FUNCTION "HF3_CP340_FC4301" : VOID	// FC 4301
TITLE = 配置本端所有CP340模块
//1：硬件配置 设置协议、波特率、奇偶校验位、起始地址
//2：需授权
//3：注意起始地址、DB块号（暂未填写）
VERSION : 0.1
BEGIN
NETWORK
TITLE = BA-21 电梯 H420/01(N) 672 2001~2005
      A     "Always0";
      =     L 0.0;
      BLD   103;
      A     "Always1";
      =     L 0.1;
      BLD   103;
      BLD   3;
      =     L 5.0;
      CDB;
      OPN   DI 1071;
      TAR2  LD 1;
      L     672;
      T     DIW 0;
      A     L 0.0;
      =     DIX 4.0;
      L     B#16#4A;
      T     DIB 5;
      L     31001;
      T     DIW 6;
      L     5;
      T     DIW 8;
      L     L#500;
      T     DID 10;
      A     L 0.1;
      =     DIX 14.0;
      L     2001;
      T     DIW 16;
      BLD   11;
      L     W#16#1002;
      T     LW 8;
      L     10;
      T     LW 10;
      L     30;
      T     LW 12;
      L     P#DBX 0.0;
      T     LD 14;
      L     W#16#1002;
      T     LW 18;
      L     10;
      T     LW 20;
      L     1071;
      T     LW 22;
      L     P#DBX 18.0;
      T     LD 24;
      UC    "BLKMOV";
      {     P#L 8.0, P#L 6.0, P#L 18.0 };
      BLD   11;
      L     W#16#1002;
      T     LW 8;
      L     10;
      T     LW 10;
      L     30;
      T     LW 12;
      L     P#DBX 10.0;
      T     LD 14;
      L     W#16#1002;
      T     LW 18;
      L     10;
      T     LW 20;
      L     1071;
      T     LW 22;
      L     P#DBX 28.0;
      T     LD 24;
      UC    "BLKMOV";
      {     P#L 8.0, P#L 6.0, P#L 18.0 };
      LAR2  P#DBX 0.0;
      UC    "MODMAS_STEP7_CP340_L";
      LAR2  LD 1;
      A     DIX 38.0;
      =     M 10.0;
      L     DIW 40;
      T     MW 12;
      L     DIW 42;
      T     MW 14;
      CDB;
      BLD   4;
      NOP   0;
NETWORK
TITLE = BA-21 局部排水泵 AP-PSB-B 688  2011~2015
      A     "Always0";
      =     L 0.0;
      BLD   103;
      A     "Always1";
      =     L 0.1;
      BLD   103;
      BLD   3;
      =     L 5.0;
      CDB;
      OPN   DI 1072;
      TAR2  LD 1;
      L     688;
      T     DIW 0;
      A     L 0.0;
      =     DIX 4.0;
      L     B#16#4A;
      T     DIB 5;
      L     31001;
      T     DIW 6;
      L     5;
      T     DIW 8;
      L     L#500;
      T     DID 10;
      A     L 0.1;
      =     DIX 14.0;
      L     2011;
      T     DIW 16;
      BLD   11;
      L     W#16#1002;
      T     LW 8;
      L     10;
      T     LW 10;
      L     30;
      T     LW 12;
      L     P#DBX 0.0;
      T     LD 14;
      L     W#16#1002;
      T     LW 18;
      L     10;
      T     LW 20;
      L     1072;
      T     LW 22;
      L     P#DBX 18.0;
      T     LD 24;
      UC    "BLKMOV";
      {     P#L 8.0, P#L 6.0, P#L 18.0 };
      BLD   11;
      L     W#16#1002;
      T     LW 8;
      L     10;
      T     LW 10;
      L     30;
      T     LW 12;
      L     P#DBX 10.0;
      T     LD 14;
      L     W#16#1002;
      T     LW 18;
      L     10;
      T     LW 20;
      L     1072;
      T     LW 22;
      L     P#DBX 28.0;
      T     LD 24;
      UC    "BLKMOV";
      {     P#L 8.0, P#L 6.0, P#L 18.0 };
      LAR2  P#DBX 0.0;
      UC    "MODMAS_STEP7_CP340_L";
      LAR2  LD 1;
      A     DIX 38.0;
      =     M 10.0;
      L     DIW 40;
      T     MW 12;
      L     DIW 42;
      T     MW 14;
      CDB;
      BLD   4;
      NOP   0;
NETWORK
TITLE = BA-21 自动扶梯 E420/05(K2)，E420/06(K2) 704 2021~2025
      A     "Always0";
      =     L 0.0;
      BLD   103;
      A     "Always1";
      =     L 0.1;
      BLD   103;
      BLD   3;
      =     L 5.0;
      CDB;
      OPN   DI 1073;
      TAR2  LD 1;
      L     704;
      T     DIW 0;
      A     L 0.0;
      =     DIX 4.0;
      L     B#16#4A;
      T     DIB 5;
      L     31001;
      T     DIW 6;
      L     5;
      T     DIW 8;
      L     L#500;
      T     DID 10;
      A     L 0.1;
      =     DIX 14.0;
      L     2021;
      T     DIW 16;
      BLD   11;
      L     W#16#1002;
      T     LW 8;
      L     10;
      T     LW 10;
      L     30;
      T     LW 12;
      L     P#DBX 0.0;
      T     LD 14;
      L     W#16#1002;
      T     LW 18;
      L     10;
      T     LW 20;
      L     1073;
      T     LW 22;
      L     P#DBX 18.0;
      T     LD 24;
      UC    "BLKMOV";
      {     P#L 8.0, P#L 6.0, P#L 18.0 };
      BLD   11;
      L     W#16#1002;
      T     LW 8;
      L     10;
      T     LW 10;
      L     30;
      T     LW 12;
      L     P#DBX 10.0;
      T     LD 14;
      L     W#16#1002;
      T     LW 18;
      L     10;
      T     LW 20;
      L     1073;
      T     LW 22;
      L     P#DBX 28.0;
      T     LD 24;
      UC    "BLKMOV";
      {     P#L 8.0, P#L 6.0, P#L 18.0 };
      LAR2  P#DBX 0.0;
      UC    "MODMAS_STEP7_CP340_L";
      LAR2  LD 1;
      A     DIX 38.0;
      =     M 10.0;
      L     DIW 40;
      T     MW 12;
      L     DIW 42;
      T     MW 14;
      CDB;
      BLD   4;
      NOP   0;
NETWORK
TITLE = BA-21 不间断电源 UPS-1 720 2031~2035
      A     "Always0";
      =     L 0.0;
      BLD   103;
      A     "Always1";
      =     L 0.1;
      BLD   103;
      BLD   3;
      =     L 5.0;
      CDB;
      OPN   DI 1074;
      TAR2  LD 1;
      L     720;
      T     DIW 0;
      A     L 0.0;
      =     DIX 4.0;
      L     B#16#4A;
      T     DIB 5;
      L     31001;
      T     DIW 6;
      L     5;
      T     DIW 8;
      L     L#500;
      T     DID 10;
      A     L 0.1;
      =     DIX 14.0;
      L     2031;
      T     DIW 16;
      BLD   11;
      L     W#16#1002;
      T     LW 8;
      L     10;
      T     LW 10;
      L     30;
      T     LW 12;
      L     P#DBX 0.0;
      T     LD 14;
      L     W#16#1002;
      T     LW 18;
      L     10;
      T     LW 20;
      L     1074;
      T     LW 22;
      L     P#DBX 18.0;
      T     LD 24;
      UC    "BLKMOV";
      {     P#L 8.0, P#L 6.0, P#L 18.0 };
      BLD   11;
      L     W#16#1002;
      T     LW 8;
      L     10;
      T     LW 10;
      L     30;
      T     LW 12;
      L     P#DBX 10.0;
      T     LD 14;
      L     W#16#1002;
      T     LW 18;
      L     10;
      T     LW 20;
      L     1074;
      T     LW 22;
      L     P#DBX 28.0;
      T     LD 24;
      UC    "BLKMOV";
      {     P#L 8.0, P#L 6.0, P#L 18.0 };
      LAR2  P#DBX 0.0;
      UC    "MODMAS_STEP7_CP340_L";
      LAR2  LD 1;
      A     DIX 38.0;
      =     M 10.0;
      L     DIW 40;
      T     MW 12;
      L     DIW 42;
      T     MW 14;
      CDB;
      BLD   4;
      NOP   0;
NETWORK
TITLE = BA-22 应急照明 EPS21 736 2041~2045
      A     "Always0";
      =     L 0.0;
      BLD   103;
      A     "Always1";
      =     L 0.1;
      BLD   103;
      BLD   3;
      =     L 5.0;
      CDB;
      OPN   DI 1075;
      TAR2  LD 1;
      L     736;
      T     DIW 0;
      A     L 0.0;
      =     DIX 4.0;
      L     B#16#4A;
      T     DIB 5;
      L     31001;
      T     DIW 6;
      L     5;
      T     DIW 8;
      L     L#500;
      T     DID 10;
      A     L 0.1;
      =     DIX 14.0;
      L     2041;
      T     DIW 16;
      BLD   11;
      L     W#16#1002;
      T     LW 8;
      L     10;
      T     LW 10;
      L     30;
      T     LW 12;
      L     P#DBX 0.0;
      T     LD 14;
      L     W#16#1002;
      T     LW 18;
      L     10;
      T     LW 20;
      L     1075;
      T     LW 22;
      L     P#DBX 18.0;
      T     LD 24;
      UC    "BLKMOV";
      {     P#L 8.0, P#L 6.0, P#L 18.0 };
      BLD   11;
      L     W#16#1002;
      T     LW 8;
      L     10;
      T     LW 10;
      L     30;
      T     LW 12;
      L     P#DBX 10.0;
      T     LD 14;
      L     W#16#1002;
      T     LW 18;
      L     10;
      T     LW 20;
      L     1075;
      T     LW 22;
      L     P#DBX 28.0;
      T     LD 24;
      UC    "BLKMOV";
      {     P#L 8.0, P#L 6.0, P#L 18.0 };
      LAR2  P#DBX 0.0;
      UC    "MODMAS_STEP7_CP340_L";
      LAR2  LD 1;
      A     DIX 38.0;
      =     M 10.0;
      L     DIW 40;
      T     MW 12;
      L     DIW 42;
      T     MW 14;
      CDB;
      BLD   4;
      NOP   0;
NETWORK
TITLE = BA-22 雨水泵 AT-AYSB1，AT-AYSB2 752 2051~2055
      A     "Always0";
      =     L 0.0;
      BLD   103;
      A     "Always1";
      =     L 0.1;
      BLD   103;
      BLD   3;
      =     L 5.0;
      CDB;
      OPN   DI 1076;
      TAR2  LD 1;
      L     752;
      T     DIW 0;
      A     L 0.0;
      =     DIX 4.0;
      L     B#16#4A;
      T     DIB 5;
      L     31001;
      T     DIW 6;
      L     5;
      T     DIW 8;
      L     L#500;
      T     DID 10;
      A     L 0.1;
      =     DIX 14.0;
      L     2051;
      T     DIW 16;
      BLD   11;
      L     W#16#1002;
      T     LW 8;
      L     10;
      T     LW 10;
      L     30;
      T     LW 12;
      L     P#DBX 0.0;
      T     LD 14;
      L     W#16#1002;
      T     LW 18;
      L     10;
      T     LW 20;
      L     1076;
      T     LW 22;
      L     P#DBX 18.0;
      T     LD 24;
      UC    "BLKMOV";
      {     P#L 8.0, P#L 6.0, P#L 18.0 };
      BLD   11;
      L     W#16#1002;
      T     LW 8;
      L     10;
      T     LW 10;
      L     30;
      T     LW 12;
      L     P#DBX 10.0;
      T     LD 14;
      L     W#16#1002;
      T     LW 18;
      L     10;
      T     LW 20;
      L     1076;
      T     LW 22;
      L     P#DBX 28.0;
      T     LD 24;
      UC    "BLKMOV";
      {     P#L 8.0, P#L 6.0, P#L 18.0 };
      LAR2  P#DBX 0.0;
      UC    "MODMAS_STEP7_CP340_L";
      LAR2  LD 1;
      A     DIX 38.0;
      =     M 10.0;
      L     DIW 40;
      T     MW 12;
      L     DIW 42;
      T     MW 14;
      CDB;
      BLD   4;
      NOP   0;
NETWORK
TITLE = BA-22 雨水泵 AT-AYSB3，AT-AYSB4，AP-FSB2 768  2061~2065
      A     "Always0";
      =     L 0.0;
      BLD   103;
      A     "Always1";
      =     L 0.1;
      BLD   103;
      BLD   3;
      =     L 5.0;
      CDB;
      OPN   DI 1077;
      TAR2  LD 1;
      L     768;
      T     DIW 0;
      A     L 0.0;
      =     DIX 4.0;
      L     B#16#4A;
      T     DIB 5;
      L     31001;
      T     DIW 6;
      L     5;
      T     DIW 8;
      L     L#500;
      T     DID 10;
      A     L 0.1;
      =     DIX 14.0;
      L     2061;
      T     DIW 16;
      BLD   11;
      L     W#16#1002;
      T     LW 8;
      L     10;
      T     LW 10;
      L     30;
      T     LW 12;
      L     P#DBX 0.0;
      T     LD 14;
      L     W#16#1002;
      T     LW 18;
      L     10;
      T     LW 20;
      L     1077;
      T     LW 22;
      L     P#DBX 18.0;
      T     LD 24;
      UC    "BLKMOV";
      {     P#L 8.0, P#L 6.0, P#L 18.0 };
      BLD   11;
      L     W#16#1002;
      T     LW 8;
      L     10;
      T     LW 10;
      L     30;
      T     LW 12;
      L     P#DBX 10.0;
      T     LD 14;
      L     W#16#1002;
      T     LW 18;
      L     10;
      T     LW 20;
      L     1077;
      T     LW 22;
      L     P#DBX 28.0;
      T     LD 24;
      UC    "BLKMOV";
      {     P#L 8.0, P#L 6.0, P#L 18.0 };
      LAR2  P#DBX 0.0;
      UC    "MODMAS_STEP7_CP340_L";
      LAR2  LD 1;
      A     DIX 38.0;
      =     M 10.0;
      L     DIW 40;
      T     MW 12;
      L     DIW 42;
      T     MW 14;
      CDB;
      BLD   4;
      NOP   0;
NETWORK
TITLE = BA-22 局排废水泵 AP-PSB-C 784 2071~2075
      A     "Always0";
      =     L 0.0;
      BLD   103;
      A     "Always1";
      =     L 0.1;
      BLD   103;
      BLD   3;
      =     L 5.0;
      CDB;
      OPN   DI 1078;
      TAR2  LD 1;
      L     784;
      T     DIW 0;
      A     L 0.0;
      =     DIX 4.0;
      L     B#16#4A;
      T     DIB 5;
      L     31001;
      T     DIW 6;
      L     5;
      T     DIW 8;
      L     L#500;
      T     DID 10;
      A     L 0.1;
      =     DIX 14.0;
      L     2071;
      T     DIW 16;
      BLD   11;
      L     W#16#1002;
      T     LW 8;
      L     10;
      T     LW 10;
      L     30;
      T     LW 12;
      L     P#DBX 0.0;
      T     LD 14;
      L     W#16#1002;
      T     LW 18;
      L     10;
      T     LW 20;
      L     1078;
      T     LW 22;
      L     P#DBX 18.0;
      T     LD 24;
      UC    "BLKMOV";
      {     P#L 8.0, P#L 6.0, P#L 18.0 };
      BLD   11;
      L     W#16#1002;
      T     LW 8;
      L     10;
      T     LW 10;
      L     30;
      T     LW 12;
      L     P#DBX 10.0;
      T     LD 14;
      L     W#16#1002;
      T     LW 18;
      L     10;
      T     LW 20;
      L     1078;
      T     LW 22;
      L     P#DBX 28.0;
      T     LD 24;
      UC    "BLKMOV";
      {     P#L 8.0, P#L 6.0, P#L 18.0 };
      LAR2  P#DBX 0.0;
      UC    "MODMAS_STEP7_CP340_L";
      LAR2  LD 1;
      A     DIX 38.0;
      =     M 10.0;
      L     DIW 40;
      T     MW 12;
      L     DIW 42;
      T     MW 14;
      CDB;
      BLD   4;
      NOP   0;
NETWORK
TITLE = BA-22 自动扶梯 E420/07(K3) 800 2081~2085
      A     "Always0";
      =     L 0.0;
      BLD   103;
      A     "Always1";
      =     L 0.1;
      BLD   103;
      BLD   3;
      =     L 5.0;
      CDB;
      OPN   DI 1079;
      TAR2  LD 1;
      L     800;
      T     DIW 0;
      A     L 0.0;
      =     DIX 4.0;
      L     B#16#4A;
      T     DIB 5;
      L     31001;
      T     DIW 6;
      L     5;
      T     DIW 8;
      L     L#500;
      T     DID 10;
      A     L 0.1;
      =     DIX 14.0;
      L     2081;
      T     DIW 16;
      BLD   11;
      L     W#16#1002;
      T     LW 8;
      L     10;
      T     LW 10;
      L     30;
      T     LW 12;
      L     P#DBX 0.0;
      T     LD 14;
      L     W#16#1002;
      T     LW 18;
      L     10;
      T     LW 20;
      L     1079;
      T     LW 22;
      L     P#DBX 18.0;
      T     LD 24;
      UC    "BLKMOV";
      {     P#L 8.0, P#L 6.0, P#L 18.0 };
      BLD   11;
      L     W#16#1002;
      T     LW 8;
      L     10;
      T     LW 10;
      L     30;
      T     LW 12;
      L     P#DBX 10.0;
      T     LD 14;
      L     W#16#1002;
      T     LW 18;
      L     10;
      T     LW 20;
      L     1079;
      T     LW 22;
      L     P#DBX 28.0;
      T     LD 24;
      UC    "BLKMOV";
      {     P#L 8.0, P#L 6.0, P#L 18.0 };
      LAR2  P#DBX 0.0;
      UC    "MODMAS_STEP7_CP340_L";
      LAR2  LD 1;
      A     DIX 38.0;
      =     M 10.0;
      L     DIW 40;
      T     MW 12;
      L     DIW 42;
      T     MW 14;
      CDB;
      BLD   4;
      NOP   0;
NETWORK
TITLE = BA-11 应急照明 EPS11 816 2091~2095
      A     "Always0";
      =     L 0.0;
      BLD   103;
      A     "Always1";
      =     L 0.1;
      BLD   103;
      BLD   3;
      =     L 5.0;
      CDB;
      OPN   DI 1080;
      TAR2  LD 1;
      L     816;
      T     DIW 0;
      A     L 0.0;
      =     DIX 4.0;
      L     B#16#4A;
      T     DIB 5;
      L     31001;
      T     DIW 6;
      L     5;
      T     DIW 8;
      L     L#500;
      T     DID 10;
      A     L 0.1;
      =     DIX 14.0;
      L     2091;
      T     DIW 16;
      BLD   11;
      L     W#16#1002;
      T     LW 8;
      L     10;
      T     LW 10;
      L     30;
      T     LW 12;
      L     P#DBX 0.0;
      T     LD 14;
      L     W#16#1002;
      T     LW 18;
      L     10;
      T     LW 20;
      L     1080;
      T     LW 22;
      L     P#DBX 18.0;
      T     LD 24;
      UC    "BLKMOV";
      {     P#L 8.0, P#L 6.0, P#L 18.0 };
      BLD   11;
      L     W#16#1002;
      T     LW 8;
      L     10;
      T     LW 10;
      L     30;
      T     LW 12;
      L     P#DBX 10.0;
      T     LD 14;
      L     W#16#1002;
      T     LW 18;
      L     10;
      T     LW 20;
      L     1080;
      T     LW 22;
      L     P#DBX 28.0;
      T     LD 24;
      UC    "BLKMOV";
      {     P#L 8.0, P#L 6.0, P#L 18.0 };
      LAR2  P#DBX 0.0;
      UC    "MODMAS_STEP7_CP340_L";
      LAR2  LD 1;
      A     DIX 38.0;
      =     M 10.0;
      L     DIW 40;
      T     MW 12;
      L     DIW 42;
      T     MW 14;
      CDB;
      BLD   4;
      NOP   0;
NETWORK
TITLE = BA-11 自动扶梯 E420/01(N) 832 2101~2105
      A     "Always0";
      =     L 0.0;
      BLD   103;
      A     "Always1";
      =     L 0.1;
      BLD   103;
      BLD   3;
      =     L 5.0;
      CDB;
      OPN   DI 1081;
      TAR2  LD 1;
      L     832;
      T     DIW 0;
      A     L 0.0;
      =     DIX 4.0;
      L     B#16#4A;
      T     DIB 5;
      L     31001;
      T     DIW 6;
      L     5;
      T     DIW 8;
      L     L#500;
      T     DID 10;
      A     L 0.1;
      =     DIX 14.0;
      L     2101;
      T     DIW 16;
      BLD   11;
      L     W#16#1002;
      T     LW 8;
      L     10;
      T     LW 10;
      L     30;
      T     LW 12;
      L     P#DBX 0.0;
      T     LD 14;
      L     W#16#1002;
      T     LW 18;
      L     10;
      T     LW 20;
      L     1081;
      T     LW 22;
      L     P#DBX 18.0;
      T     LD 24;
      UC    "BLKMOV";
      {     P#L 8.0, P#L 6.0, P#L 18.0 };
      BLD   11;
      L     W#16#1002;
      T     LW 8;
      L     10;
      T     LW 10;
      L     30;
      T     LW 12;
      L     P#DBX 10.0;
      T     LD 14;
      L     W#16#1002;
      T     LW 18;
      L     10;
      T     LW 20;
      L     1081;
      T     LW 22;
      L     P#DBX 28.0;
      T     LD 24;
      UC    "BLKMOV";
      {     P#L 8.0, P#L 6.0, P#L 18.0 };
      LAR2  P#DBX 0.0;
      UC    "MODMAS_STEP7_CP340_L";
      LAR2  LD 1;
      A     DIX 38.0;
      =     M 10.0;
      L     DIW 40;
      T     MW 12;
      L     DIW 42;
      T     MW 14;
      CDB;
      BLD   4;
      NOP   0;
NETWORK
TITLE = BQ11 区间水泵 ATD-HSB 944 2181~2185
      A     "Always0";
      =     L 0.0;
      BLD   103;
      A     "Always1";
      =     L 0.1;
      BLD   103;
      BLD   3;
      =     L 5.0;
      CDB;
      OPN   DI 1082;
      TAR2  LD 1;
      L     944;
      T     DIW 0;
      A     L 0.0;
      =     DIX 4.0;
      L     B#16#4A;
      T     DIB 5;
      L     31001;
      T     DIW 6;
      L     5;
      T     DIW 8;
      L     L#500;
      T     DID 10;
      A     L 0.1;
      =     DIX 14.0;
      L     2181;
      T     DIW 16;
      BLD   11;
      L     W#16#1002;
      T     LW 8;
      L     10;
      T     LW 10;
      L     30;
      T     LW 12;
      L     P#DBX 0.0;
      T     LD 14;
      L     W#16#1002;
      T     LW 18;
      L     10;
      T     LW 20;
      L     1082;
      T     LW 22;
      L     P#DBX 18.0;
      T     LD 24;
      UC    "BLKMOV";
      {     P#L 8.0, P#L 6.0, P#L 18.0 };
      BLD   11;
      L     W#16#1002;
      T     LW 8;
      L     10;
      T     LW 10;
      L     30;
      T     LW 12;
      L     P#DBX 10.0;
      T     LD 14;
      L     W#16#1002;
      T     LW 18;
      L     10;
      T     LW 20;
      L     1082;
      T     LW 22;
      L     P#DBX 28.0;
      T     LD 24;
      UC    "BLKMOV";
      {     P#L 8.0, P#L 6.0, P#L 18.0 };
      LAR2  P#DBX 0.0;
      UC    "MODMAS_STEP7_CP340_L";
      LAR2  LD 1;
      A     DIX 38.0;
      =     M 10.0;
      L     DIW 40;
      T     MW 12;
      L     DIW 42;
      T     MW 14;
      CDB;
      BLD   4;
      NOP   0;
END_FUNCTION

DATA_BLOCK "CONTROL_DAT"	// DB 1
VERSION : 0.1
  STRUCT
   id_0_a : WORD ;
   id_1_a : WORD ;
   reuse_conn_time : TIME ;
   use_all_conn : BOOL ;
   RECV_TIMEOUT : TIME ;
   CONN_TIMEOUT : TIME ;
   DISCONNECT : BOOL ;
   Init : BOOL ;
   ENQ : BOOL ;
   DATA_TYPE : BYTE ;
   START_ADDRESS : WORD ;
   LENGTH : WORD ;
   WRITE_READ : BOOL ;
   UNIT : BYTE  := B#16#1;
   LICENSED : BOOL ;
   BUSY : BOOL ;
   DONE : BOOL ;
   ERROR : BOOL ;
   ESTAB_0A : BOOL ;
   STATUS_0A : WORD ;
   ESTAB_1A : BOOL ;
   STATUS_1A : WORD ;
   RedErrS7 : BOOL ;
   RedErrDev : BOOL ;
   TotComErr : BOOL ;
   Init_Error : BOOL ;
   Init_Status : WORD ;
   Save_STATUS_0A : WORD ;
   Save_STATUS_1A : WORD ;
   Count_Done : DINT ;
   Count_Error : DINT ;
  END_STRUCT ;	
BEGIN
   UNIT := B#16#1;
END_DATA_BLOCK

DATA_BLOCK "MODBUS_HPARAM_PN_2"	// DB 2
TITLE = Parameters for Modbus TCP
AUTHOR : SIEMENS
FAMILY : COMM
NAME : MBHPARAM
VERSION : 0.1
  STRUCT
   double_sided_red : BOOL ;
   connection_0A : STRUCT
    block_length : WORD  := W#16#40;	//#!Verbindung_0001!#
    id : WORD  := W#16#1;
    connection_type : BYTE  := B#16#11;
    active_est : BOOL  := TRUE;
    local_device_id : BYTE  := B#16#5;
    local_tsap_id_len : BYTE ;
    rem_subnet_id_len : BYTE ;
    rem_staddr_len : BYTE  := B#16#4;
    rem_tsap_id_len : BYTE  := B#16#2;
    next_staddr_len : BYTE ;
    local_tsap_id : ARRAY  [1 .. 16 ] OF BYTE  := 16 (B#16#0) ;
    rem_subnet_id : ARRAY  [1 .. 6 ] OF BYTE  := B#16#0, B#16#0, B#16#0, B#16#0, B#16#0, B#16#0;
    rem_staddr : ARRAY  [1 .. 6 ] OF BYTE  := B#16#A, B#16#2E, B#16#1E, B#16#97;
    rem_tsap_id : ARRAY  [1 .. 16 ] OF BYTE  := B#16#1, B#16#F6;
    next_staddr : ARRAY  [1 .. 6 ] OF BYTE  := B#16#0, B#16#0, B#16#0, B#16#0, B#16#0, B#16#0;
    spare : WORD ;	//#!Verbindung_0001!#
   END_STRUCT ;
   connection_1A : STRUCT
    block_length : WORD  := W#16#40;	//#!Verbindung_0002!#
    id : WORD  := W#16#2;
    connection_type : BYTE  := B#16#11;
    active_est : BOOL  := TRUE;
    local_device_id : BYTE  := B#16#15;
    local_tsap_id_len : BYTE ;
    rem_subnet_id_len : BYTE ;
    rem_staddr_len : BYTE  := B#16#4;
    rem_tsap_id_len : BYTE  := B#16#2;
    next_staddr_len : BYTE ;
    local_tsap_id : ARRAY  [1 .. 16 ] OF BYTE  := 16 (B#16#0) ;
    rem_subnet_id : ARRAY  [1 .. 6 ] OF BYTE  := B#16#0, B#16#0, B#16#0, B#16#0, B#16#0, B#16#0;
    rem_staddr : ARRAY  [1 .. 6 ] OF BYTE  := B#16#A, B#16#2E, B#16#82, B#16#97;
    rem_tsap_id : ARRAY  [1 .. 16 ] OF BYTE  := B#16#1, B#16#F6;
    next_staddr : ARRAY  [1 .. 6 ] OF BYTE  := B#16#0, B#16#0, B#16#0, B#16#0, B#16#0, B#16#0;
    spare : WORD ;	//#!Verbindung_0002!#
   END_STRUCT ;
   server_client : BOOL ;
   single_write : BOOL ;
   connect_at_startup : BOOL  := TRUE;
   reserved : BYTE ;
   data_type_1 : BYTE  := B#16#3;
   db_1 : WORD  := W#16#8F3;
   start_1 : WORD ;
   end_1 : WORD  := W#16#18F;
   data_type_2 : BYTE  := B#16#3;
   db_2 : WORD  := W#16#8F4;
   start_2 : WORD  := W#16#190;
   end_2 : WORD  := W#16#22F;
   data_type_3 : BYTE ;
   db_3 : WORD  := W#16#D;
   start_3 : WORD  := W#16#2D0;
   end_3 : WORD  := W#16#3E8;
   data_type_4 : BYTE ;
   db_4 : WORD ;
   start_4 : WORD ;
   end_4 : WORD ;
   data_type_5 : BYTE ;
   db_5 : WORD  := W#16#E;
   start_5 : WORD  := W#16#280;
   end_5 : WORD  := W#16#4E2;
   data_type_6 : BYTE ;
   db_6 : WORD  := W#16#F;
   start_6 : WORD  := W#16#6A4;
   end_6 : WORD  := W#16#8FC;
   data_type_7 : BYTE ;
   db_7 : WORD  := W#16#10;
   start_7 : WORD  := W#16#6A4;
   end_7 : WORD  := W#16#8FC;
   data_type_8 : BYTE ;
   db_8 : WORD ;
   start_8 : WORD ;
   end_8 : WORD ;
   conn_0A_send_buffer : ARRAY  [1 .. 260 ] OF BYTE  := 260 (B#16#0) ;
   conn_0A_recv_buffer : ARRAY  [1 .. 260 ] OF BYTE  := 260 (B#16#0) ;
   conn_1A_send_buffer : ARRAY  [1 .. 260 ] OF BYTE  := 260 (B#16#0) ;
   conn_1A_recv_buffer : ARRAY  [1 .. 260 ] OF BYTE  := 260 (B#16#0) ;
  END_STRUCT ;	
BEGIN
   connection_0A.block_length := W#16#40;
   connection_0A.id := W#16#1;
   connection_0A.connection_type := B#16#11;
   connection_0A.active_est := TRUE;
   connection_0A.local_device_id := B#16#5;
   connection_0A.rem_staddr_len := B#16#4;
   connection_0A.rem_tsap_id_len := B#16#2;
   connection_0A.rem_staddr[1] := B#16#A;
   connection_0A.rem_staddr[2] := B#16#2E;
   connection_0A.rem_staddr[3] := B#16#1E;
   connection_0A.rem_staddr[4] := B#16#97;
   connection_0A.rem_tsap_id[1] := B#16#1;
   connection_0A.rem_tsap_id[2] := B#16#F6;
   connection_1A.block_length := W#16#40;
   connection_1A.id := W#16#2;
   connection_1A.connection_type := B#16#11;
   connection_1A.active_est := TRUE;
   connection_1A.local_device_id := B#16#15;
   connection_1A.rem_staddr_len := B#16#4;
   connection_1A.rem_tsap_id_len := B#16#2;
   connection_1A.rem_staddr[1] := B#16#A;
   connection_1A.rem_staddr[2] := B#16#2E;
   connection_1A.rem_staddr[3] := B#16#82;
   connection_1A.rem_staddr[4] := B#16#97;
   connection_1A.rem_tsap_id[1] := B#16#1;
   connection_1A.rem_tsap_id[2] := B#16#F6;
   connect_at_startup := TRUE;
   data_type_1 := B#16#3;
   db_1 := W#16#8F3;
   end_1 := W#16#18F;
   data_type_2 := B#16#3;
   db_2 := W#16#8F4;
   start_2 := W#16#190;
   end_2 := W#16#22F;
   db_3 := W#16#D;
   start_3 := W#16#2D0;
   end_3 := W#16#3E8;
   db_5 := W#16#E;
   start_5 := W#16#280;
   end_5 := W#16#4E2;
   db_6 := W#16#F;
   start_6 := W#16#6A4;
   end_6 := W#16#8FC;
   db_7 := W#16#10;
   start_7 := W#16#6A4;
   end_7 := W#16#8FC;
END_DATA_BLOCK

DATA_BLOCK "License DB"	// DB 3
VERSION : 0.1
  STRUCT
   REG_KEY : STRING  [17 ] := 'insert REG_KEY';	//Registration Key
  END_STRUCT ;	
BEGIN
   REG_KEY := 'insert REG_KEY';
END_DATA_BLOCK

DATA_BLOCK DB 10
VERSION : 0.1
  STRUCT
   DB_VAR1 : REAL  := 6.700000e+000;	//Temporary placeholder variable
   DB_VAR2 : REAL ;
  END_STRUCT ;	
BEGIN
END_DATA_BLOCK

DATA_BLOCK DB 12
VERSION : 0.1
  STRUCT
   DB_VAR : ARRAY  [0 .. 76 ] OF //Holding Register 3001-3077
   WORD  := 77 (W#16#0) ;
   reserved : WORD ;
  END_STRUCT ;	
BEGIN
END_DATA_BLOCK

DATA_BLOCK "CPULINDB"	// DB 30
VERSION : 0.1
  STRUCT
   YOULIN1 : STRING  [8 ] := 'R1R3H5Y4';	//Temporary placeholder variable
   YOULIN2 : STRING  [8 ] := '3N5L1J32';
  END_STRUCT ;	
BEGIN
   YOULIN1 := 'R1R3H5Y4';
   YOULIN2 := '3N5L1J32';
END_DATA_BLOCK

DATA_BLOCK "SYS_Date_Time_D"	// DB 34
VERSION : 0.1
  STRUCT
   SET_DATE_TIME : ARRAY  [1 .. 8 ] OF //年月日时分秒
   BYTE ;
   READ_DATE_TIME : ARRAY  [1 .. 8 ] OF BYTE ;
   SET : DATE_AND_TIME ;
   READ : DATE_AND_TIME ;
   TIME_HM : INT ;	//时分(2359表示23点59分)
  END_STRUCT ;	
BEGIN
END_DATA_BLOCK

DATA_BLOCK "FB200_DB"	// DB 200
VERSION : 0.0
"S7400H-COM-MAIN-SLAVE"
BEGIN
END_DATA_BLOCK

DATA_BLOCK "FB201_DB"	// DB 201
VERSION : 0.0
"S7400H-COM-MAIN-IBP"
BEGIN
END_DATA_BLOCK

DATA_BLOCK "MAIN-READ-SLAVE"	// DB 202
VERSION : 0.1
  STRUCT
   MAIN_R_SLAVE : ARRAY  [0 .. 4000 ] OF //Temporary placeholder variable
   INT  := 0;
  END_STRUCT ;	
BEGIN
END_DATA_BLOCK

DATA_BLOCK "MAIN-WRITE-SLAVE"	// DB 203
VERSION : 0.1
  STRUCT
   MAIN_W_SLAVE : ARRAY  [0 .. 4000 ] OF //Temporary placeholder variable
   INT  := 0;
  END_STRUCT ;	
BEGIN
END_DATA_BLOCK

DATA_BLOCK "MAIN-READ-IBP"	// DB 204
VERSION : 0.1
  STRUCT
   MAIN_R_IBP : ARRAY  [0 .. 4000 ] OF //Temporary placeholder variable
   INT  := 0;
  END_STRUCT ;	
BEGIN
END_DATA_BLOCK

DATA_BLOCK "MAIN-WRITE-IBP"	// DB 205
VERSION : 0.1
  STRUCT
   MAIN_W_IBP : ARRAY  [0 .. 4000 ] OF //Temporary placeholder variable
   INT  := 0;
  END_STRUCT ;	
BEGIN
END_DATA_BLOCK

DATA_BLOCK "DETAIL_DIAG_DB_RACK0"	// DB 458
AUTHOR : SIEMENS
FAMILY : DP
VERSION : 0.1
"DETAIL_DP_DIAG"
BEGIN
END_DATA_BLOCK

DATA_BLOCK "DETAIL_DIAG_DB_RACK1"	// DB 459
AUTHOR : SIEMENS
FAMILY : DP
VERSION : 0.1
"DETAIL_DP_DIAG"
BEGIN
END_DATA_BLOCK

DATA_BLOCK "DP_ERROR_RACK0"	// DB 460
VERSION : 0.1
  STRUCT
   STATE : ARRAY  [0 .. 500 ] OF //Temporary placeholder variable
   INT ;
   STATE_NONE : ARRAY  [0 .. 50 ] OF INT ;
   ALL_OK : BOOL ;
   TIME_RESET : BOOL ;
   NOTUSED : ARRAY  [0 .. 250 ] OF INT ;
  END_STRUCT ;	
BEGIN
END_DATA_BLOCK

DATA_BLOCK "DP_ERROR_RESET_DB"	// DB 461
VERSION : 0.1
  STRUCT
   STATE : ARRAY  [0 .. 500 ] OF //Temporary placeholder variable
   INT ;
   STATE_NONE : ARRAY  [0 .. 50 ] OF INT ;
   ALL_OK : BOOL ;
   TIME_RESET : BOOL ;
   NOTUSED : ARRAY  [0 .. 250 ] OF INT ;
  END_STRUCT ;	
BEGIN
END_DATA_BLOCK

DATA_BLOCK "DP_ERROR_FB1501"	// DB 462
VERSION : 0.0
"com_check"
BEGIN
END_DATA_BLOCK

DATA_BLOCK "DB_FOR_FB300"	// DB 463
VERSION : 0.1
"READ_ERROR"
BEGIN
END_DATA_BLOCK

DATA_BLOCK "DP_VAT"	// DB 464
VERSION : 0.1
  STRUCT
   MANUAL_MODE : BOOL ;
   SINGLE_STEP_SLAVE : BOOL ;
   SINGLE_STEP_ERROR : BOOL ;
   RESET : BOOL ;
   SINGLE_SLAVE_DIAG : BOOL ;
   SINGLE_DIAG_ADR : BYTE ;
   ALL_SLAVES_OK : BOOL ;
   SUM_SLAVES_DIAG : BYTE ;
   SLAVE_ADR : BYTE ;
   SLAVE_STATE : BYTE ;
   SLAVE_IDENT_NO : WORD ;
   ERROR_NO : BYTE ;
   ERROR_TYPE : BYTE ;
   MODULE_NO : BYTE ;
   MODULE_STATE : BYTE ;
   CHANNEL_NO : BYTE ;
   CHANNEL_TYPE : BYTE ;
   CHANNEL_ERROR_CODE : INT ;
   CHANNEL_ERROR_INFO_1 : DWORD ;
   CHANNEL_ERROR_INFO_2 : DWORD ;
   DIAG_COUNTER : BYTE ;
   DIAG_OVERFLOW : BOOL ;
   BUSY : BOOL ;
   MANUAL_MODE1 : BOOL ;
   SINGLE_STEP_SLAVE1 : BOOL ;
   SINGLE_STEP_ERROR1 : BOOL ;
   RESET1 : BOOL ;
   SINGLE_SLAVE_DIAG1 : BOOL ;
   SINGLE_DIAG_ADR1 : BYTE ;
   ALL_SLAVES_OK1 : BOOL ;
   SUM_SLAVES_DIAG1 : BYTE ;
   SLAVE_ADR1 : BYTE ;
   SLAVE_STATE1 : BYTE ;
   SLAVE_IDENT_NO1 : WORD ;
   ERROR_NO1 : BYTE ;
   ERROR_TYPE1 : BYTE ;
   MODULE_NO1 : BYTE ;
   MODULE_STATE1 : BYTE ;
   CHANNEL_NO1 : BYTE ;
   CHANNEL_TYPE1 : BYTE ;
   CHANNEL_ERROR_CODE1 : INT ;
   CHANNEL_ERROR_INFO_11 : DWORD ;
   CHANNEL_ERROR_INFO_21 : DWORD ;
   DIAG_COUNTER1 : BYTE ;
   DIAG_OVERFLOW1 : BOOL ;
   BUSY1 : BOOL ;
   TIME_RESET : BOOL ;
  END_STRUCT ;	
BEGIN
END_DATA_BLOCK

DATA_BLOCK "DP_ERROR_RACK1"	// DB 465
VERSION : 0.1
  STRUCT
   STATE : ARRAY  [0 .. 500 ] OF //Temporary placeholder variable
   INT ;
   STATE_NONE : ARRAY  [0 .. 50 ] OF INT ;
   ALL_OK : BOOL ;
   TIME_RESET : BOOL ;
   NOTUSED : ARRAY  [0 .. 250 ] OF INT ;
  END_STRUCT ;	
BEGIN
END_DATA_BLOCK

DATA_BLOCK "DP_ERROR1_RESET"	// DB 466
VERSION : 0.1
  STRUCT
   STATE : ARRAY  [0 .. 500 ] OF //Temporary placeholder variable
   INT ;
   STATE_NONE : ARRAY  [0 .. 50 ] OF INT ;
   ALL_OK : BOOL ;
   TIME_RESET : BOOL ;
   NOTUSED : ARRAY  [0 .. 250 ] OF INT ;
  END_STRUCT ;	
BEGIN
END_DATA_BLOCK

DATA_BLOCK "DP_ERROR1_FB1501"	// DB 467
VERSION : 0.0
"com_check"
BEGIN
END_DATA_BLOCK

DATA_BLOCK "FB523_DB"	// DB 523
AUTHOR : KNAB
FAMILY : DIAGNOSE
VERSION : 0.0
"H_STATUS"
BEGIN
END_DATA_BLOCK

DATA_BLOCK "LED"	// DB 525
VERSION : 0.1
  STRUCT
   EXTF : ARRAY  [0 .. 8 ] OF BYTE ;
   REDF : ARRAY  [0 .. 8 ] OF BYTE ;
   EXTF_RET_VAL : INT ;
   REDF_RET_VAL : INT ;
   EXTF_BUSY : BOOL ;
   REDF_BUSY : BOOL ;
  END_STRUCT ;	
BEGIN
END_DATA_BLOCK

DATA_BLOCK DB 777
VERSION : 0.0
"HF4_IMCC_TVF_FB2652"
BEGIN
END_DATA_BLOCK

DATA_BLOCK "IDB_MODBUS"	// DB 915
AUTHOR : SIEMENS
FAMILY : COMM
VERSION : 0.0
"MB_PNHCL"
BEGIN
END_DATA_BLOCK

DATA_BLOCK "JOBLIST_DB"	// DB 919
AUTHOR : SIEMENS
FAMILY : COMM
VERSION : 0.0
"Job_List"
BEGIN
END_DATA_BLOCK

DATA_BLOCK "JOB_RESET_DB"	// DB 921
VERSION : 0.0
"JOB_RESET"
BEGIN
END_DATA_BLOCK

DATA_BLOCK DB 1072
AUTHOR : Dixinke
FAMILY : ASCMOD
VERSION : 0.0
"MODMAS_STEP7_CP340_L"
BEGIN
END_DATA_BLOCK

DATA_BLOCK DB 1073
AUTHOR : Dixinke
FAMILY : ASCMOD
VERSION : 0.0
"MODMAS_STEP7_CP340_L"
BEGIN
END_DATA_BLOCK

DATA_BLOCK DB 1074
AUTHOR : Dixinke
FAMILY : ASCMOD
VERSION : 0.0
"MODMAS_STEP7_CP340_L"
BEGIN
END_DATA_BLOCK

DATA_BLOCK DB 1075
AUTHOR : Dixinke
FAMILY : ASCMOD
VERSION : 0.0
"MODMAS_STEP7_CP340_L"
BEGIN
END_DATA_BLOCK

DATA_BLOCK DB 1076
AUTHOR : Dixinke
FAMILY : ASCMOD
VERSION : 0.0
"MODMAS_STEP7_CP340_L"
BEGIN
END_DATA_BLOCK

DATA_BLOCK DB 1077
AUTHOR : Dixinke
FAMILY : ASCMOD
VERSION : 0.0
"MODMAS_STEP7_CP340_L"
BEGIN
END_DATA_BLOCK

DATA_BLOCK DB 1078
AUTHOR : Dixinke
FAMILY : ASCMOD
VERSION : 0.0
"MODMAS_STEP7_CP340_L"
BEGIN
END_DATA_BLOCK

DATA_BLOCK DB 1079
AUTHOR : Dixinke
FAMILY : ASCMOD
VERSION : 0.0
"MODMAS_STEP7_CP340_L"
BEGIN
END_DATA_BLOCK

DATA_BLOCK DB 1080
AUTHOR : Dixinke
FAMILY : ASCMOD
VERSION : 0.0
"MODMAS_STEP7_CP340_L"
BEGIN
END_DATA_BLOCK

DATA_BLOCK DB 1081
AUTHOR : Dixinke
FAMILY : ASCMOD
VERSION : 0.0
"MODMAS_STEP7_CP340_L"
BEGIN
END_DATA_BLOCK

DATA_BLOCK DB 1082
AUTHOR : Dixinke
FAMILY : ASCMOD
VERSION : 0.0
"MODMAS_STEP7_CP340_L"
BEGIN
END_DATA_BLOCK

DATA_BLOCK DB 2000
VERSION : 0.1
  STRUCT
   DB_VAR : ARRAY  [0 .. 194 ] OF //Holding Register 2001-2195
   WORD  := 195 (W#16#0) ;
   reserved : WORD ;
  END_STRUCT ;	
BEGIN
END_DATA_BLOCK

DATA_BLOCK DB 2001
VERSION : 0.0
  STRUCT
   START_SEQ : BYTE  := B#16#1;
   END_SEQ : BYTE  := B#16#1;
   SND_COMM_DB : WORD  := W#16#7D2;
   WRT_COMM_DB : WORD  := W#16#7D3;
   WRT_COMP_DB : WORD  := W#16#7D4;
   DAT_RECV_DB : WORD  := W#16#7D5;
   ACT_1 : BOOL  := TRUE;
   Mode_1 : BOOL ;
   SND_DB_1 : INT  := 2002;
   SND_ADD_1 : INT ;
   SND_LEN_1 : INT  := 6;
   RCV_DB_1 : INT  := 2005;
   RCV_ADD_1 : INT ;
   RCV_LEN_1 : INT  := 10;
   WD_TIME_1 : INT  := 3000;
   VBVer : WORD  := W#16#29;	//配置文件版本号
  END_STRUCT ;	
BEGIN
   START_SEQ := B#16#1;
   END_SEQ := B#16#1;
   SND_COMM_DB := W#16#7D2;
   WRT_COMM_DB := W#16#7D3;
   WRT_COMP_DB := W#16#7D4;
   DAT_RECV_DB := W#16#7D5;
   ACT_1 := TRUE;
   SND_DB_1 := 2002;
   SND_LEN_1 := 6;
   RCV_DB_1 := 2005;
   RCV_LEN_1 := 10;
   WD_TIME_1 := 3000;
   VBVer := W#16#29;
END_DATA_BLOCK

DATA_BLOCK DB 2002
VERSION : 0.0
  STRUCT
   SlaveID_1 : BYTE  := B#16#B;
   FC_1 : BYTE  := B#16#3;
   START_ADD_1 : WORD ;
   DATA_NUM_1 : WORD  := W#16#4;
   CRC_1 : WORD ;
  END_STRUCT ;	
BEGIN
   SlaveID_1 := B#16#B;
   FC_1 := B#16#3;
   DATA_NUM_1 := W#16#4;
END_DATA_BLOCK

DATA_BLOCK "AP_BMPSB"	// DB 2005
VERSION : 0.0
  STRUCT
   Command_1_STATUS : WORD ;	//第1条命令的状态，0=正常，1=无响应，2=站号错误，3=命令错误，4=CRC校验错误
   Command_1_DATA_1 : WORD ;	//地址40001
   Command_1_DATA_2 : WORD ;	//地址40002
   Command_1_DATA_3 : WORD ;	//地址40003
   Command_1_DATA_4 : WORD ;	//地址40004
  END_STRUCT ;	
BEGIN
END_DATA_BLOCK

DATA_BLOCK DB 2011
VERSION : 0.0
  STRUCT
   START_SEQ : BYTE  := B#16#1;
   END_SEQ : BYTE  := B#16#1;
   SND_COMM_DB : WORD  := W#16#7DC;
   WRT_COMM_DB : WORD  := W#16#7DD;
   WRT_COMP_DB : WORD  := W#16#7DE;
   DAT_RECV_DB : WORD  := W#16#7DF;
   ACT_1 : BOOL  := TRUE;
   Mode_1 : BOOL ;
   SND_DB_1 : INT  := 2012;
   SND_ADD_1 : INT ;
   SND_LEN_1 : INT  := 6;
   RCV_DB_1 : INT  := 2015;
   RCV_ADD_1 : INT ;
   RCV_LEN_1 : INT  := 36;
   WD_TIME_1 : INT  := 3000;
   VBVer : WORD  := W#16#29;	//配置文件版本号
  END_STRUCT ;	
BEGIN
   START_SEQ := B#16#1;
   END_SEQ := B#16#1;
   SND_COMM_DB := W#16#7DC;
   WRT_COMM_DB := W#16#7DD;
   WRT_COMP_DB := W#16#7DE;
   DAT_RECV_DB := W#16#7DF;
   ACT_1 := TRUE;
   SND_DB_1 := 2012;
   SND_LEN_1 := 6;
   RCV_DB_1 := 2015;
   RCV_LEN_1 := 36;
   WD_TIME_1 := 3000;
   VBVer := W#16#29;
END_DATA_BLOCK

DATA_BLOCK DB 2012
VERSION : 0.0
  STRUCT
   SlaveID_1 : BYTE  := B#16#B;
   FC_1 : BYTE  := B#16#3;
   START_ADD_1 : WORD ;
   DATA_NUM_1 : WORD  := W#16#11;
   CRC_1 : WORD ;
  END_STRUCT ;	
BEGIN
   SlaveID_1 := B#16#B;
   FC_1 := B#16#3;
   DATA_NUM_1 := W#16#11;
END_DATA_BLOCK

DATA_BLOCK "EPS21"	// DB 2015
VERSION : 0.0
  STRUCT
   Command_1_STATUS : WORD ;	//第1条命令的状态，0=正常，1=无响应，2=站号错误，3=命令错误，4=CRC校验错误
   Command_1_DATA_1 : WORD ;	//地址40001
   Command_1_DATA_2 : WORD ;	//地址40002
   Command_1_DATA_3 : WORD ;	//地址40003
   Command_1_DATA_4 : WORD ;	//地址40004
   Command_1_DATA_5 : WORD ;	//地址40005
   Command_1_DATA_6 : WORD ;	//地址40006
   Command_1_DATA_7 : WORD ;	//地址40007
   Command_1_DATA_8 : WORD ;	//地址40008
   Command_1_DATA_9 : WORD ;	//地址40009
   Command_1_DATA_10 : WORD ;	//地址40010
   Command_1_DATA_11 : WORD ;	//地址40011
   Command_1_DATA_12 : WORD ;	//地址40012
   Command_1_DATA_13 : WORD ;	//地址40013
   Command_1_DATA_14 : WORD ;	//地址40014
   Command_1_DATA_15 : WORD ;	//地址40015
   Command_1_DATA_16 : WORD ;	//地址40016
   Command_1_DATA_17 : WORD ;	//地址40017
  END_STRUCT ;	
BEGIN
END_DATA_BLOCK

DATA_BLOCK DB 2021
VERSION : 0.0
  STRUCT
   START_SEQ : BYTE  := B#16#1;
   END_SEQ : BYTE  := B#16#2;
   SND_COMM_DB : WORD  := W#16#7E6;
   WRT_COMM_DB : WORD  := W#16#7E7;
   WRT_COMP_DB : WORD  := W#16#7E8;
   DAT_RECV_DB : WORD  := W#16#7E9;
   ACT_1 : BOOL  := TRUE;
   Mode_1 : BOOL ;
   SND_DB_1 : INT  := 2022;
   SND_ADD_1 : INT ;
   SND_LEN_1 : INT  := 6;
   RCV_DB_1 : INT  := 2025;
   RCV_ADD_1 : INT ;
   RCV_LEN_1 : INT  := 4;
   WD_TIME_1 : INT  := 3000;
   ACT_2 : BOOL  := TRUE;
   Mode_2 : BOOL ;
   SND_DB_2 : INT  := 2022;
   SND_ADD_2 : INT  := 8;
   SND_LEN_2 : INT  := 6;
   RCV_DB_2 : INT  := 2025;
   RCV_ADD_2 : INT  := 4;
   RCV_LEN_2 : INT  := 4;
   WD_TIME_2 : INT  := 3000;
   VBVer : WORD  := W#16#29;	//配置文件版本号
  END_STRUCT ;	
BEGIN
   START_SEQ := B#16#1;
   END_SEQ := B#16#2;
   SND_COMM_DB := W#16#7E6;
   WRT_COMM_DB := W#16#7E7;
   WRT_COMP_DB := W#16#7E8;
   DAT_RECV_DB := W#16#7E9;
   ACT_1 := TRUE;
   SND_DB_1 := 2022;
   SND_LEN_1 := 6;
   RCV_DB_1 := 2025;
   RCV_LEN_1 := 4;
   WD_TIME_1 := 3000;
   ACT_2 := TRUE;
   SND_DB_2 := 2022;
   SND_ADD_2 := 8;
   SND_LEN_2 := 6;
   RCV_DB_2 := 2025;
   RCV_ADD_2 := 4;
   RCV_LEN_2 := 4;
   WD_TIME_2 := 3000;
   VBVer := W#16#29;
END_DATA_BLOCK

DATA_BLOCK DB 2022
VERSION : 0.0
  STRUCT
   SlaveID_1 : BYTE  := B#16#B;
   FC_1 : BYTE  := B#16#3;
   START_ADD_1 : WORD  := W#16#1;
   DATA_NUM_1 : WORD  := W#16#1;
   CRC_1 : WORD ;
   SlaveID_2 : BYTE  := B#16#B;
   FC_2 : BYTE  := B#16#3;
   START_ADD_2 : WORD  := W#16#14;
   DATA_NUM_2 : WORD  := W#16#1;
   CRC_2 : WORD ;
  END_STRUCT ;	
BEGIN
   SlaveID_1 := B#16#B;
   FC_1 := B#16#3;
   START_ADD_1 := W#16#1;
   DATA_NUM_1 := W#16#1;
   SlaveID_2 := B#16#B;
   FC_2 := B#16#3;
   START_ADD_2 := W#16#14;
   DATA_NUM_2 := W#16#1;
END_DATA_BLOCK

DATA_BLOCK "E411_08_C"	// DB 2025
VERSION : 0.0
  STRUCT
   Command_1_STATUS : WORD ;	//第1条命令的状态，0=正常，1=无响应，2=站号错误，3=命令错误，4=CRC校验错误
   Command_1_DATA_1 : WORD ;	//地址40002
   Command_2_STATUS : WORD ;	//第2条命令的状态，0=正常，1=无响应，2=站号错误，3=命令错误，4=CRC校验错误
   Command_2_DATA_1 : WORD ;	//地址40021
  END_STRUCT ;	
BEGIN
END_DATA_BLOCK

DATA_BLOCK DB 2031
VERSION : 0.0
  STRUCT
   START_SEQ : BYTE  := B#16#1;
   END_SEQ : BYTE  := B#16#5;
   SND_COMM_DB : WORD  := W#16#7F0;
   WRT_COMM_DB : WORD  := W#16#7F1;
   WRT_COMP_DB : WORD  := W#16#7F2;
   DAT_RECV_DB : WORD  := W#16#7F3;
   ACT_1 : BOOL  := TRUE;
   Mode_1 : BOOL ;
   SND_DB_1 : INT  := 2032;
   SND_ADD_1 : INT ;
   SND_LEN_1 : INT  := 6;
   RCV_DB_1 : INT  := 2035;
   RCV_ADD_1 : INT ;
   RCV_LEN_1 : INT  := 10;
   WD_TIME_1 : INT  := 3000;
   ACT_2 : BOOL  := TRUE;
   Mode_2 : BOOL ;
   SND_DB_2 : INT  := 2034;
   SND_ADD_2 : INT ;
   SND_LEN_2 : INT  := 10;
   RCV_DB_2 : INT  := 2035;
   RCV_ADD_2 : INT  := 10;
   RCV_LEN_2 : INT  := 2;
   WD_TIME_2 : INT  := 3000;
   ACT_3 : BOOL  := TRUE;
   Mode_3 : BOOL ;
   SND_DB_3 : INT  := 2032;
   SND_ADD_3 : INT  := 8;
   SND_LEN_3 : INT  := 6;
   RCV_DB_3 : INT  := 2035;
   RCV_ADD_3 : INT  := 12;
   RCV_LEN_3 : INT  := 10;
   WD_TIME_3 : INT  := 3000;
   ACT_4 : BOOL  := TRUE;
   Mode_4 : BOOL ;
   SND_DB_4 : INT  := 2034;
   SND_ADD_4 : INT  := 12;
   SND_LEN_4 : INT  := 10;
   RCV_DB_4 : INT  := 2035;
   RCV_ADD_4 : INT  := 22;
   RCV_LEN_4 : INT  := 2;
   WD_TIME_4 : INT  := 3000;
   ACT_5 : BOOL  := TRUE;
   Mode_5 : BOOL ;
   SND_DB_5 : INT  := 2032;
   SND_ADD_5 : INT  := 16;
   SND_LEN_5 : INT  := 6;
   RCV_DB_5 : INT  := 2035;
   RCV_ADD_5 : INT  := 24;
   RCV_LEN_5 : INT  := 10;
   WD_TIME_5 : INT  := 3000;
   VBVer : WORD  := W#16#2B;	//配置文件版本号
  END_STRUCT ;	
BEGIN
   START_SEQ := B#16#1;
   END_SEQ := B#16#5;
   SND_COMM_DB := W#16#7F0;
   WRT_COMM_DB := W#16#7F1;
   WRT_COMP_DB := W#16#7F2;
   DAT_RECV_DB := W#16#7F3;
   ACT_1 := TRUE;
   SND_DB_1 := 2032;
   SND_LEN_1 := 6;
   RCV_DB_1 := 2035;
   RCV_LEN_1 := 10;
   WD_TIME_1 := 3000;
   ACT_2 := TRUE;
   SND_DB_2 := 2034;
   SND_LEN_2 := 10;
   RCV_DB_2 := 2035;
   RCV_ADD_2 := 10;
   RCV_LEN_2 := 2;
   WD_TIME_2 := 3000;
   ACT_3 := TRUE;
   SND_DB_3 := 2032;
   SND_ADD_3 := 8;
   SND_LEN_3 := 6;
   RCV_DB_3 := 2035;
   RCV_ADD_3 := 12;
   RCV_LEN_3 := 10;
   WD_TIME_3 := 3000;
   ACT_4 := TRUE;
   SND_DB_4 := 2034;
   SND_ADD_4 := 12;
   SND_LEN_4 := 10;
   RCV_DB_4 := 2035;
   RCV_ADD_4 := 22;
   RCV_LEN_4 := 2;
   WD_TIME_4 := 3000;
   ACT_5 := TRUE;
   SND_DB_5 := 2032;
   SND_ADD_5 := 16;
   SND_LEN_5 := 6;
   RCV_DB_5 := 2035;
   RCV_ADD_5 := 24;
   RCV_LEN_5 := 10;
   WD_TIME_5 := 3000;
   VBVer := W#16#2B;
END_DATA_BLOCK

DATA_BLOCK DB 2032
VERSION : 0.0
  STRUCT
   SlaveID_1 : BYTE  := B#16#B;
   FC_1 : BYTE  := B#16#3;
   START_ADD_1 : WORD ;
   DATA_NUM_1 : WORD  := W#16#4;
   CRC_1 : WORD ;
   SlaveID_3 : BYTE  := B#16#C;
   FC_3 : BYTE  := B#16#3;
   START_ADD_3 : WORD ;
   DATA_NUM_3 : WORD  := W#16#4;
   CRC_3 : WORD ;
   SlaveID_5 : BYTE  := B#16#D;
   FC_5 : BYTE  := B#16#3;
   START_ADD_5 : WORD ;
   DATA_NUM_5 : WORD  := W#16#4;
   CRC_5 : WORD ;
  END_STRUCT ;	
BEGIN
   SlaveID_1 := B#16#B;
   FC_1 := B#16#3;
   DATA_NUM_1 := W#16#4;
   SlaveID_3 := B#16#C;
   FC_3 := B#16#3;
   DATA_NUM_3 := W#16#4;
   SlaveID_5 := B#16#D;
   FC_5 := B#16#3;
   DATA_NUM_5 := W#16#4;
END_DATA_BLOCK

DATA_BLOCK "AT_AYSB4_WRITE"	// DB 2033
VERSION : 0.0
  STRUCT
   SlaveID_2 : BYTE  := B#16#B;
   FC_2 : BYTE  := B#16#10;
   START_ADD_2 : WORD  := W#16#4;
   DATA_NUM_2 : WORD  := W#16#1;
   DATA_BYTE_2 : WORD  := W#16#2;
   DATA_2_1 : WORD ;	//地址40005
   CRC_2 : WORD ;
   SlaveID_4 : BYTE  := B#16#C;
   FC_4 : BYTE  := B#16#10;
   START_ADD_4 : WORD  := W#16#4;
   DATA_NUM_4 : WORD  := W#16#1;
   DATA_BYTE_4 : WORD  := W#16#2;
   DATA_4_1 : WORD ;	//地址40005
   CRC_4 : WORD ;
  END_STRUCT ;	
BEGIN
   SlaveID_2 := B#16#B;
   FC_2 := B#16#10;
   START_ADD_2 := W#16#4;
   DATA_NUM_2 := W#16#1;
   DATA_BYTE_2 := W#16#2;
   SlaveID_4 := B#16#C;
   FC_4 := B#16#10;
   START_ADD_4 := W#16#4;
   DATA_NUM_4 := W#16#1;
   DATA_BYTE_4 := W#16#2;
END_DATA_BLOCK

DATA_BLOCK DB 2034
VERSION : 0.0
  STRUCT
   SlaveID_2 : BYTE  := B#16#B;
   FC_2 : BYTE  := B#16#10;
   START_ADD_2 : WORD  := W#16#4;
   DATA_NUM_2 : WORD  := W#16#1;
   DATA_BYTE_2 : WORD  := W#16#2;
   DATA_NUM_2_1 : WORD ;
   CRC_2 : WORD ;
   SlaveID_4 : BYTE  := B#16#C;
   FC_4 : BYTE  := B#16#10;
   START_ADD_4 : WORD  := W#16#4;
   DATA_NUM_4 : WORD  := W#16#1;
   DATA_BYTE_4 : WORD  := W#16#2;
   DATA_NUM_4_1 : WORD ;
   CRC_4 : WORD ;
  END_STRUCT ;	
BEGIN
   SlaveID_2 := B#16#B;
   FC_2 := B#16#10;
   START_ADD_2 := W#16#4;
   DATA_NUM_2 := W#16#1;
   DATA_BYTE_2 := W#16#2;
   SlaveID_4 := B#16#C;
   FC_4 := B#16#10;
   START_ADD_4 := W#16#4;
   DATA_NUM_4 := W#16#1;
   DATA_BYTE_4 := W#16#2;
END_DATA_BLOCK

DATA_BLOCK "AT_AYSB4_READ"	// DB 2035
VERSION : 0.0
  STRUCT
   Command_1_STATUS : WORD ;	//第1条命令的状态，0=正常，1=无响应，2=站号错误，3=命令错误，4=CRC校验错误
   Command_1_DATA_1 : WORD ;	//地址40001
   Command_1_DATA_2 : WORD ;	//地址40002
   Command_1_DATA_3 : WORD ;	//地址40003
   Command_1_DATA_4 : WORD ;	//地址40004
   Command_2_STATUS : WORD ;	//第2条命令的状态，0=正常，1=无响应，2=站号错误，3=命令错误，4=CRC校验错误
   Command_3_STATUS : WORD ;	//第3条命令的状态，0=正常，1=无响应，2=站号错误，3=命令错误，4=CRC校验错误
   Command_3_DATA_1 : WORD ;	//地址40001
   Command_3_DATA_2 : WORD ;	//地址40002
   Command_3_DATA_3 : WORD ;	//地址40003
   Command_3_DATA_4 : WORD ;	//地址40004
   Command_4_STATUS : WORD ;	//第4条命令的状态，0=正常，1=无响应，2=站号错误，3=命令错误，4=CRC校验错误
   Command_5_STATUS : WORD ;	//第5条命令的状态，0=正常，1=无响应，2=站号错误，3=命令错误，4=CRC校验错误
   Command_5_DATA_1 : WORD ;	//地址40001
   Command_5_DATA_2 : WORD ;	//地址40002
   Command_5_DATA_3 : WORD ;	//地址40003
   Command_5_DATA_4 : WORD ;	//地址40004
  END_STRUCT ;	
BEGIN
END_DATA_BLOCK

DATA_BLOCK DB 2041
VERSION : 0.0
  STRUCT
   START_SEQ : BYTE  := B#16#1;
   END_SEQ : BYTE  := B#16#4;
   SND_COMM_DB : WORD  := W#16#7FA;
   WRT_COMM_DB : WORD  := W#16#7FB;
   WRT_COMP_DB : WORD  := W#16#7FC;
   DAT_RECV_DB : WORD  := W#16#7FD;
   ACT_1 : BOOL  := TRUE;
   Mode_1 : BOOL ;
   SND_DB_1 : INT  := 2042;
   SND_ADD_1 : INT ;
   SND_LEN_1 : INT  := 6;
   RCV_DB_1 : INT  := 2045;
   RCV_ADD_1 : INT ;
   RCV_LEN_1 : INT  := 10;
   WD_TIME_1 : INT  := 3000;
   ACT_2 : BOOL  := TRUE;
   Mode_2 : BOOL ;
   SND_DB_2 : INT  := 2044;
   SND_ADD_2 : INT ;
   SND_LEN_2 : INT  := 10;
   RCV_DB_2 : INT  := 2045;
   RCV_ADD_2 : INT  := 10;
   RCV_LEN_2 : INT  := 2;
   WD_TIME_2 : INT  := 3000;
   ACT_3 : BOOL  := TRUE;
   Mode_3 : BOOL ;
   SND_DB_3 : INT  := 2042;
   SND_ADD_3 : INT  := 8;
   SND_LEN_3 : INT  := 6;
   RCV_DB_3 : INT  := 2045;
   RCV_ADD_3 : INT  := 12;
   RCV_LEN_3 : INT  := 10;
   WD_TIME_3 : INT  := 3000;
   ACT_4 : BOOL  := TRUE;
   Mode_4 : BOOL ;
   SND_DB_4 : INT  := 2044;
   SND_ADD_4 : INT  := 12;
   SND_LEN_4 : INT  := 10;
   RCV_DB_4 : INT  := 2045;
   RCV_ADD_4 : INT  := 22;
   RCV_LEN_4 : INT  := 2;
   WD_TIME_4 : INT  := 3000;
   VBVer : WORD  := W#16#2B;	//配置文件版本号
  END_STRUCT ;	
BEGIN
   START_SEQ := B#16#1;
   END_SEQ := B#16#4;
   SND_COMM_DB := W#16#7FA;
   WRT_COMM_DB := W#16#7FB;
   WRT_COMP_DB := W#16#7FC;
   DAT_RECV_DB := W#16#7FD;
   ACT_1 := TRUE;
   SND_DB_1 := 2042;
   SND_LEN_1 := 6;
   RCV_DB_1 := 2045;
   RCV_LEN_1 := 10;
   WD_TIME_1 := 3000;
   ACT_2 := TRUE;
   SND_DB_2 := 2044;
   SND_LEN_2 := 10;
   RCV_DB_2 := 2045;
   RCV_ADD_2 := 10;
   RCV_LEN_2 := 2;
   WD_TIME_2 := 3000;
   ACT_3 := TRUE;
   SND_DB_3 := 2042;
   SND_ADD_3 := 8;
   SND_LEN_3 := 6;
   RCV_DB_3 := 2045;
   RCV_ADD_3 := 12;
   RCV_LEN_3 := 10;
   WD_TIME_3 := 3000;
   ACT_4 := TRUE;
   SND_DB_4 := 2044;
   SND_ADD_4 := 12;
   SND_LEN_4 := 10;
   RCV_DB_4 := 2045;
   RCV_ADD_4 := 22;
   RCV_LEN_4 := 2;
   WD_TIME_4 := 3000;
   VBVer := W#16#2B;
END_DATA_BLOCK

DATA_BLOCK DB 2042
VERSION : 0.0
  STRUCT
   SlaveID_1 : BYTE  := B#16#B;
   FC_1 : BYTE  := B#16#3;
   START_ADD_1 : WORD ;
   DATA_NUM_1 : WORD  := W#16#4;
   CRC_1 : WORD ;
   SlaveID_3 : BYTE  := B#16#C;
   FC_3 : BYTE  := B#16#3;
   START_ADD_3 : WORD ;
   DATA_NUM_3 : WORD  := W#16#4;
   CRC_3 : WORD ;
  END_STRUCT ;	
BEGIN
   SlaveID_1 := B#16#B;
   FC_1 := B#16#3;
   DATA_NUM_1 := W#16#4;
   SlaveID_3 := B#16#C;
   FC_3 := B#16#3;
   DATA_NUM_3 := W#16#4;
END_DATA_BLOCK

DATA_BLOCK "AT_aysb1_2_WRITE"	// DB 2043
VERSION : 0.0
  STRUCT
   SlaveID_2 : BYTE  := B#16#B;
   FC_2 : BYTE  := B#16#10;
   START_ADD_2 : WORD  := W#16#4;
   DATA_NUM_2 : WORD  := W#16#1;
   DATA_BYTE_2 : WORD  := W#16#2;
   DATA_2_1 : WORD ;	//地址40005
   CRC_2 : WORD ;
   SlaveID_4 : BYTE  := B#16#C;
   FC_4 : BYTE  := B#16#10;
   START_ADD_4 : WORD  := W#16#4;
   DATA_NUM_4 : WORD  := W#16#1;
   DATA_BYTE_4 : WORD  := W#16#2;
   DATA_4_1 : WORD ;	//地址40005
   CRC_4 : WORD ;
  END_STRUCT ;	
BEGIN
   SlaveID_2 := B#16#B;
   FC_2 := B#16#10;
   START_ADD_2 := W#16#4;
   DATA_NUM_2 := W#16#1;
   DATA_BYTE_2 := W#16#2;
   SlaveID_4 := B#16#C;
   FC_4 := B#16#10;
   START_ADD_4 := W#16#4;
   DATA_NUM_4 := W#16#1;
   DATA_BYTE_4 := W#16#2;
END_DATA_BLOCK

DATA_BLOCK DB 2044
VERSION : 0.0
  STRUCT
   SlaveID_2 : BYTE  := B#16#B;
   FC_2 : BYTE  := B#16#10;
   START_ADD_2 : WORD  := W#16#4;
   DATA_NUM_2 : WORD  := W#16#1;
   DATA_BYTE_2 : WORD  := W#16#2;
   DATA_NUM_2_1 : WORD ;
   CRC_2 : WORD ;
   SlaveID_4 : BYTE  := B#16#C;
   FC_4 : BYTE  := B#16#10;
   START_ADD_4 : WORD  := W#16#4;
   DATA_NUM_4 : WORD  := W#16#1;
   DATA_BYTE_4 : WORD  := W#16#2;
   DATA_NUM_4_1 : WORD ;
   CRC_4 : WORD ;
  END_STRUCT ;	
BEGIN
   SlaveID_2 := B#16#B;
   FC_2 := B#16#10;
   START_ADD_2 := W#16#4;
   DATA_NUM_2 := W#16#1;
   DATA_BYTE_2 := W#16#2;
   SlaveID_4 := B#16#C;
   FC_4 := B#16#10;
   START_ADD_4 := W#16#4;
   DATA_NUM_4 := W#16#1;
   DATA_BYTE_4 := W#16#2;
END_DATA_BLOCK

DATA_BLOCK "AT_AYSB1_2_READ"	// DB 2045
VERSION : 0.0
  STRUCT
   Command_1_STATUS : WORD ;	//第1条命令的状态，0=正常，1=无响应，2=站号错误，3=命令错误，4=CRC校验错误
   Command_1_DATA_1 : WORD ;	//地址40001
   Command_1_DATA_2 : WORD ;	//地址40002
   Command_1_DATA_3 : WORD ;	//地址40003
   Command_1_DATA_4 : WORD ;	//地址40004
   Command_2_STATUS : WORD ;	//第2条命令的状态，0=正常，1=无响应，2=站号错误，3=命令错误，4=CRC校验错误
   Command_3_STATUS : WORD ;	//第3条命令的状态，0=正常，1=无响应，2=站号错误，3=命令错误，4=CRC校验错误
   Command_3_DATA_1 : WORD ;	//地址40001
   Command_3_DATA_2 : WORD ;	//地址40002
   Command_3_DATA_3 : WORD ;	//地址40003
   Command_3_DATA_4 : WORD ;	//地址40004
   Command_4_STATUS : WORD ;	//第4条命令的状态，0=正常，1=无响应，2=站号错误，3=命令错误，4=CRC校验错误
  END_STRUCT ;	
BEGIN
END_DATA_BLOCK

DATA_BLOCK DB 2051
VERSION : 0.0
  STRUCT
   START_SEQ : BYTE  := B#16#1;
   END_SEQ : BYTE  := B#16#2;
   SND_COMM_DB : WORD  := W#16#804;
   WRT_COMM_DB : WORD  := W#16#805;
   WRT_COMP_DB : WORD  := W#16#806;
   DAT_RECV_DB : WORD  := W#16#807;
   ACT_1 : BOOL  := TRUE;
   Mode_1 : BOOL ;
   SND_DB_1 : INT  := 2052;
   SND_ADD_1 : INT ;
   SND_LEN_1 : INT  := 6;
   RCV_DB_1 : INT  := 2055;
   RCV_ADD_1 : INT ;
   RCV_LEN_1 : INT  := 10;
   WD_TIME_1 : INT  := 3000;
   ACT_2 : BOOL  := TRUE;
   Mode_2 : BOOL ;
   SND_DB_2 : INT  := 2052;
   SND_ADD_2 : INT  := 8;
   SND_LEN_2 : INT  := 6;
   RCV_DB_2 : INT  := 2055;
   RCV_ADD_2 : INT  := 10;
   RCV_LEN_2 : INT  := 10;
   WD_TIME_2 : INT  := 3000;
   VBVer : WORD  := W#16#29;	//配置文件版本号
  END_STRUCT ;	
BEGIN
   START_SEQ := B#16#1;
   END_SEQ := B#16#2;
   SND_COMM_DB := W#16#804;
   WRT_COMM_DB := W#16#805;
   WRT_COMP_DB := W#16#806;
   DAT_RECV_DB := W#16#807;
   ACT_1 := TRUE;
   SND_DB_1 := 2052;
   SND_LEN_1 := 6;
   RCV_DB_1 := 2055;
   RCV_LEN_1 := 10;
   WD_TIME_1 := 3000;
   ACT_2 := TRUE;
   SND_DB_2 := 2052;
   SND_ADD_2 := 8;
   SND_LEN_2 := 6;
   RCV_DB_2 := 2055;
   RCV_ADD_2 := 10;
   RCV_LEN_2 := 10;
   WD_TIME_2 := 3000;
   VBVer := W#16#29;
END_DATA_BLOCK

DATA_BLOCK DB 2052
VERSION : 0.0
  STRUCT
   SlaveID_1 : BYTE  := B#16#B;
   FC_1 : BYTE  := B#16#3;
   START_ADD_1 : WORD ;
   DATA_NUM_1 : WORD  := W#16#4;
   CRC_1 : WORD ;
   SlaveID_2 : BYTE  := B#16#C;
   FC_2 : BYTE  := B#16#3;
   START_ADD_2 : WORD ;
   DATA_NUM_2 : WORD  := W#16#4;
   CRC_2 : WORD ;
  END_STRUCT ;	
BEGIN
   SlaveID_1 := B#16#B;
   FC_1 := B#16#3;
   DATA_NUM_1 := W#16#4;
   SlaveID_2 := B#16#C;
   FC_2 := B#16#3;
   DATA_NUM_2 := W#16#4;
END_DATA_BLOCK

DATA_BLOCK "AP_PSB_C1_C2"	// DB 2055
VERSION : 0.0
  STRUCT
   Command_1_STATUS : WORD ;	//第1条命令的状态，0=正常，1=无响应，2=站号错误，3=命令错误，4=CRC校验错误
   Command_1_DATA_1 : WORD ;	//地址40001
   Command_1_DATA_2 : WORD ;	//地址40002
   Command_1_DATA_3 : WORD ;	//地址40003
   Command_1_DATA_4 : WORD ;	//地址40004
   Command_2_STATUS : WORD ;	//第2条命令的状态，0=正常，1=无响应，2=站号错误，3=命令错误，4=CRC校验错误
   Command_2_DATA_1 : WORD ;	//地址40001
   Command_2_DATA_2 : WORD ;	//地址40002
   Command_2_DATA_3 : WORD ;	//地址40003
   Command_2_DATA_4 : WORD ;	//地址40004
  END_STRUCT ;	
BEGIN
END_DATA_BLOCK

DATA_BLOCK DB 2061
VERSION : 0.0
  STRUCT
   START_SEQ : BYTE  := B#16#1;
   END_SEQ : BYTE  := B#16#5;
   SND_COMM_DB : WORD  := W#16#80E;
   WRT_COMM_DB : WORD  := W#16#80F;
   WRT_COMP_DB : WORD  := W#16#810;
   DAT_RECV_DB : WORD  := W#16#811;
   ACT_1 : BOOL  := TRUE;
   Mode_1 : BOOL ;
   SND_DB_1 : INT  := 2062;
   SND_ADD_1 : INT ;
   SND_LEN_1 : INT  := 6;
   RCV_DB_1 : INT  := 2065;
   RCV_ADD_1 : INT ;
   RCV_LEN_1 : INT  := 10;
   WD_TIME_1 : INT  := 3000;
   ACT_2 : BOOL  := TRUE;
   Mode_2 : BOOL ;
   SND_DB_2 : INT  := 2064;
   SND_ADD_2 : INT ;
   SND_LEN_2 : INT  := 10;
   RCV_DB_2 : INT  := 2065;
   RCV_ADD_2 : INT  := 10;
   RCV_LEN_2 : INT  := 2;
   WD_TIME_2 : INT  := 3000;
   ACT_3 : BOOL  := TRUE;
   Mode_3 : BOOL ;
   SND_DB_3 : INT  := 2062;
   SND_ADD_3 : INT  := 8;
   SND_LEN_3 : INT  := 6;
   RCV_DB_3 : INT  := 2065;
   RCV_ADD_3 : INT  := 12;
   RCV_LEN_3 : INT  := 10;
   WD_TIME_3 : INT  := 3000;
   ACT_4 : BOOL  := TRUE;
   Mode_4 : BOOL ;
   SND_DB_4 : INT  := 2064;
   SND_ADD_4 : INT  := 12;
   SND_LEN_4 : INT  := 10;
   RCV_DB_4 : INT  := 2065;
   RCV_ADD_4 : INT  := 22;
   RCV_LEN_4 : INT  := 2;
   WD_TIME_4 : INT  := 3000;
   ACT_5 : BOOL  := TRUE;
   Mode_5 : BOOL ;
   SND_DB_5 : INT  := 2062;
   SND_ADD_5 : INT  := 16;
   SND_LEN_5 : INT  := 6;
   RCV_DB_5 : INT  := 2065;
   RCV_ADD_5 : INT  := 24;
   RCV_LEN_5 : INT  := 10;
   WD_TIME_5 : INT  := 3000;
   VBVer : WORD  := W#16#2B;	//配置文件版本号
  END_STRUCT ;	
BEGIN
   START_SEQ := B#16#1;
   END_SEQ := B#16#5;
   SND_COMM_DB := W#16#80E;
   WRT_COMM_DB := W#16#80F;
   WRT_COMP_DB := W#16#810;
   DAT_RECV_DB := W#16#811;
   ACT_1 := TRUE;
   SND_DB_1 := 2062;
   SND_LEN_1 := 6;
   RCV_DB_1 := 2065;
   RCV_LEN_1 := 10;
   WD_TIME_1 := 3000;
   ACT_2 := TRUE;
   SND_DB_2 := 2064;
   SND_LEN_2 := 10;
   RCV_DB_2 := 2065;
   RCV_ADD_2 := 10;
   RCV_LEN_2 := 2;
   WD_TIME_2 := 3000;
   ACT_3 := TRUE;
   SND_DB_3 := 2062;
   SND_ADD_3 := 8;
   SND_LEN_3 := 6;
   RCV_DB_3 := 2065;
   RCV_ADD_3 := 12;
   RCV_LEN_3 := 10;
   WD_TIME_3 := 3000;
   ACT_4 := TRUE;
   SND_DB_4 := 2064;
   SND_ADD_4 := 12;
   SND_LEN_4 := 10;
   RCV_DB_4 := 2065;
   RCV_ADD_4 := 22;
   RCV_LEN_4 := 2;
   WD_TIME_4 := 3000;
   ACT_5 := TRUE;
   SND_DB_5 := 2062;
   SND_ADD_5 := 16;
   SND_LEN_5 := 6;
   RCV_DB_5 := 2065;
   RCV_ADD_5 := 24;
   RCV_LEN_5 := 10;
   WD_TIME_5 := 3000;
   VBVer := W#16#2B;
END_DATA_BLOCK

DATA_BLOCK DB 2062
VERSION : 0.0
  STRUCT
   SlaveID_1 : BYTE  := B#16#B;
   FC_1 : BYTE  := B#16#3;
   START_ADD_1 : WORD ;
   DATA_NUM_1 : WORD  := W#16#4;
   CRC_1 : WORD ;
   SlaveID_3 : BYTE  := B#16#C;
   FC_3 : BYTE  := B#16#3;
   START_ADD_3 : WORD ;
   DATA_NUM_3 : WORD  := W#16#4;
   CRC_3 : WORD ;
   SlaveID_5 : BYTE  := B#16#D;
   FC_5 : BYTE  := B#16#3;
   START_ADD_5 : WORD ;
   DATA_NUM_5 : WORD  := W#16#4;
   CRC_5 : WORD ;
  END_STRUCT ;	
BEGIN
   SlaveID_1 := B#16#B;
   FC_1 := B#16#3;
   DATA_NUM_1 := W#16#4;
   SlaveID_3 := B#16#C;
   FC_3 := B#16#3;
   DATA_NUM_3 := W#16#4;
   SlaveID_5 := B#16#D;
   FC_5 := B#16#3;
   DATA_NUM_5 := W#16#4;
END_DATA_BLOCK

DATA_BLOCK DB 2063
VERSION : 0.0
  STRUCT
   SlaveID_2 : BYTE  := B#16#B;
   FC_2 : BYTE  := B#16#10;
   START_ADD_2 : WORD  := W#16#4;
   DATA_NUM_2 : WORD  := W#16#1;
   DATA_BYTE_2 : WORD  := W#16#2;
   DATA_2_1 : WORD ;	//地址40005
   CRC_2 : WORD ;
   SlaveID_4 : BYTE  := B#16#C;
   FC_4 : BYTE  := B#16#10;
   START_ADD_4 : WORD  := W#16#4;
   DATA_NUM_4 : WORD  := W#16#1;
   DATA_BYTE_4 : WORD  := W#16#2;
   DATA_4_1 : WORD ;	//地址40005
   CRC_4 : WORD ;
  END_STRUCT ;	
BEGIN
   SlaveID_2 := B#16#B;
   FC_2 := B#16#10;
   START_ADD_2 := W#16#4;
   DATA_NUM_2 := W#16#1;
   DATA_BYTE_2 := W#16#2;
   SlaveID_4 := B#16#C;
   FC_4 := B#16#10;
   START_ADD_4 := W#16#4;
   DATA_NUM_4 := W#16#1;
   DATA_BYTE_4 := W#16#2;
END_DATA_BLOCK

DATA_BLOCK DB 2064
VERSION : 0.0
  STRUCT
   SlaveID_2 : BYTE  := B#16#B;
   FC_2 : BYTE  := B#16#10;
   START_ADD_2 : WORD  := W#16#4;
   DATA_NUM_2 : WORD  := W#16#1;
   DATA_BYTE_2 : WORD  := W#16#2;
   DATA_NUM_2_1 : WORD ;
   CRC_2 : WORD ;
   SlaveID_4 : BYTE  := B#16#C;
   FC_4 : BYTE  := B#16#10;
   START_ADD_4 : WORD  := W#16#4;
   DATA_NUM_4 : WORD  := W#16#1;
   DATA_BYTE_4 : WORD  := W#16#2;
   DATA_NUM_4_1 : WORD ;
   CRC_4 : WORD ;
  END_STRUCT ;	
BEGIN
   SlaveID_2 := B#16#B;
   FC_2 := B#16#10;
   START_ADD_2 := W#16#4;
   DATA_NUM_2 := W#16#1;
   DATA_BYTE_2 := W#16#2;
   SlaveID_4 := B#16#C;
   FC_4 := B#16#10;
   START_ADD_4 := W#16#4;
   DATA_NUM_4 := W#16#1;
   DATA_BYTE_4 := W#16#2;
END_DATA_BLOCK

DATA_BLOCK "AT_FSB_3_4_PSD2"	// DB 2065
VERSION : 0.0
  STRUCT
   Command_1_STATUS : WORD ;	//第1条命令的状态，0=正常，1=无响应，2=站号错误，3=命令错误，4=CRC校验错误
   Command_1_DATA_1 : WORD ;	//地址40001
   Command_1_DATA_2 : WORD ;	//地址40002
   Command_1_DATA_3 : WORD ;	//地址40003
   Command_1_DATA_4 : WORD ;	//地址40004
   Command_2_STATUS : WORD ;	//第2条命令的状态，0=正常，1=无响应，2=站号错误，3=命令错误，4=CRC校验错误
   Command_3_STATUS : WORD ;	//第3条命令的状态，0=正常，1=无响应，2=站号错误，3=命令错误，4=CRC校验错误
   Command_3_DATA_1 : WORD ;	//地址40001
   Command_3_DATA_2 : WORD ;	//地址40002
   Command_3_DATA_3 : WORD ;	//地址40003
   Command_3_DATA_4 : WORD ;	//地址40004
   Command_4_STATUS : WORD ;	//第4条命令的状态，0=正常，1=无响应，2=站号错误，3=命令错误，4=CRC校验错误
   Command_5_STATUS : WORD ;	//第5条命令的状态，0=正常，1=无响应，2=站号错误，3=命令错误，4=CRC校验错误
   Command_5_DATA_1 : WORD ;	//地址40001
   Command_5_DATA_2 : WORD ;	//地址40002
   Command_5_DATA_3 : WORD ;	//地址40003
   Command_5_DATA_4 : WORD ;	//地址40004
  END_STRUCT ;	
BEGIN
END_DATA_BLOCK

DATA_BLOCK DB 2071
VERSION : 0.0
  STRUCT
   START_SEQ : BYTE  := B#16#1;
   END_SEQ : BYTE  := B#16#1;
   SND_COMM_DB : WORD  := W#16#818;
   WRT_COMM_DB : WORD  := W#16#819;
   WRT_COMP_DB : WORD  := W#16#81A;
   DAT_RECV_DB : WORD  := W#16#81B;
   ACT_1 : BOOL  := TRUE;
   Mode_1 : BOOL ;
   SND_DB_1 : INT  := 2072;
   SND_ADD_1 : INT ;
   SND_LEN_1 : INT  := 6;
   RCV_DB_1 : INT  := 2075;
   RCV_ADD_1 : INT ;
   RCV_LEN_1 : INT  := 10;
   WD_TIME_1 : INT  := 3000;
   VBVer : WORD  := W#16#2B;	//配置文件版本号
  END_STRUCT ;	
BEGIN
   START_SEQ := B#16#1;
   END_SEQ := B#16#1;
   SND_COMM_DB := W#16#818;
   WRT_COMM_DB := W#16#819;
   WRT_COMP_DB := W#16#81A;
   DAT_RECV_DB := W#16#81B;
   ACT_1 := TRUE;
   SND_DB_1 := 2072;
   SND_LEN_1 := 6;
   RCV_DB_1 := 2075;
   RCV_LEN_1 := 10;
   WD_TIME_1 := 3000;
   VBVer := W#16#2B;
END_DATA_BLOCK

DATA_BLOCK DB 2072
VERSION : 0.0
  STRUCT
   SlaveID_1 : BYTE  := B#16#B;
   FC_1 : BYTE  := B#16#3;
   START_ADD_1 : WORD ;
   DATA_NUM_1 : WORD  := W#16#4;
   CRC_1 : WORD ;
  END_STRUCT ;	
BEGIN
   SlaveID_1 := B#16#B;
   FC_1 := B#16#3;
   DATA_NUM_1 := W#16#4;
END_DATA_BLOCK

DATA_BLOCK "AP_PSB_C"	// DB 2075
VERSION : 0.0
  STRUCT
   Command_1_STATUS : WORD ;	//第1条命令的状态，0=正常，1=无响应，2=站号错误，3=命令错误，4=CRC校验错误
   Command_1_DATA_1 : WORD ;	//地址40001
   Command_1_DATA_2 : WORD ;	//地址40002
   Command_1_DATA_3 : WORD ;	//地址40003
   Command_1_DATA_4 : WORD ;	//地址40004
  END_STRUCT ;	
BEGIN
END_DATA_BLOCK

DATA_BLOCK DB 2091
VERSION : 0.0
  STRUCT
   START_SEQ : BYTE  := B#16#1;
   END_SEQ : BYTE  := B#16#1;
   SND_COMM_DB : WORD  := W#16#82C;
   WRT_COMM_DB : WORD  := W#16#82D;
   WRT_COMP_DB : WORD  := W#16#82E;
   DAT_RECV_DB : WORD  := W#16#82F;
   ACT_1 : BOOL  := TRUE;
   Mode_1 : BOOL ;
   SND_DB_1 : INT  := 2092;
   SND_ADD_1 : INT ;
   SND_LEN_1 : INT  := 6;
   RCV_DB_1 : INT  := 2095;
   RCV_ADD_1 : INT ;
   RCV_LEN_1 : INT  := 36;
   WD_TIME_1 : INT  := 3000;
   VBVer : WORD  := W#16#29;	//配置文件版本号
  END_STRUCT ;	
BEGIN
   START_SEQ := B#16#1;
   END_SEQ := B#16#1;
   SND_COMM_DB := W#16#82C;
   WRT_COMM_DB := W#16#82D;
   WRT_COMP_DB := W#16#82E;
   DAT_RECV_DB := W#16#82F;
   ACT_1 := TRUE;
   SND_DB_1 := 2092;
   SND_LEN_1 := 6;
   RCV_DB_1 := 2095;
   RCV_LEN_1 := 36;
   WD_TIME_1 := 3000;
   VBVer := W#16#29;
END_DATA_BLOCK

DATA_BLOCK DB 2092
VERSION : 0.0
  STRUCT
   SlaveID_1 : BYTE  := B#16#B;
   FC_1 : BYTE  := B#16#3;
   START_ADD_1 : WORD ;
   DATA_NUM_1 : WORD  := W#16#11;
   CRC_1 : WORD ;
  END_STRUCT ;	
BEGIN
   SlaveID_1 := B#16#B;
   FC_1 := B#16#3;
   DATA_NUM_1 := W#16#11;
END_DATA_BLOCK

DATA_BLOCK "EPS11"	// DB 2095
VERSION : 0.0
  STRUCT
   Command_1_STATUS : WORD ;	//第1条命令的状态，0=正常，1=无响应，2=站号错误，3=命令错误，4=CRC校验错误
   Command_1_DATA_1 : WORD ;	//地址40001
   Command_1_DATA_2 : WORD ;	//地址40002
   Command_1_DATA_3 : WORD ;	//地址40003
   Command_1_DATA_4 : WORD ;	//地址40004
   Command_1_DATA_5 : WORD ;	//地址40005
   Command_1_DATA_6 : WORD ;	//地址40006
   Command_1_DATA_7 : WORD ;	//地址40007
   Command_1_DATA_8 : WORD ;	//地址40008
   Command_1_DATA_9 : WORD ;	//地址40009
   Command_1_DATA_10 : WORD ;	//地址40010
   Command_1_DATA_11 : WORD ;	//地址40011
   Command_1_DATA_12 : WORD ;	//地址40012
   Command_1_DATA_13 : WORD ;	//地址40013
   Command_1_DATA_14 : WORD ;	//地址40014
   Command_1_DATA_15 : WORD ;	//地址40015
   Command_1_DATA_16 : WORD ;	//地址40016
   Command_1_DATA_17 : WORD ;	//地址40017
  END_STRUCT ;	
BEGIN
END_DATA_BLOCK

DATA_BLOCK DB 2101
VERSION : 0.0
  STRUCT
   START_SEQ : BYTE  := B#16#1;
   END_SEQ : BYTE  := B#16#1;
   SND_COMM_DB : WORD  := W#16#836;
   WRT_COMM_DB : WORD  := W#16#837;
   WRT_COMP_DB : WORD  := W#16#838;
   DAT_RECV_DB : WORD  := W#16#839;
   ACT_1 : BOOL  := TRUE;
   Mode_1 : BOOL ;
   SND_DB_1 : INT  := 2102;
   SND_ADD_1 : INT ;
   SND_LEN_1 : INT  := 6;
   RCV_DB_1 : INT  := 2105;
   RCV_ADD_1 : INT ;
   RCV_LEN_1 : INT  := 6;
   WD_TIME_1 : INT  := 3000;
   VBVer : WORD  := W#16#2B;	//配置文件版本号
  END_STRUCT ;	
BEGIN
   START_SEQ := B#16#1;
   END_SEQ := B#16#1;
   SND_COMM_DB := W#16#836;
   WRT_COMM_DB := W#16#837;
   WRT_COMP_DB := W#16#838;
   DAT_RECV_DB := W#16#839;
   ACT_1 := TRUE;
   SND_DB_1 := 2102;
   SND_LEN_1 := 6;
   RCV_DB_1 := 2105;
   RCV_LEN_1 := 6;
   WD_TIME_1 := 3000;
   VBVer := W#16#2B;
END_DATA_BLOCK

DATA_BLOCK DB 2102
VERSION : 0.0
  STRUCT
   SlaveID_1 : BYTE  := B#16#1;
   FC_1 : BYTE  := B#16#3;
   START_ADD_1 : WORD  := W#16#14;
   DATA_NUM_1 : WORD  := W#16#2;
   CRC_1 : WORD ;
  END_STRUCT ;	
BEGIN
   SlaveID_1 := B#16#1;
   FC_1 := B#16#3;
   START_ADD_1 := W#16#14;
   DATA_NUM_1 := W#16#2;
END_DATA_BLOCK

DATA_BLOCK "E411_01_02_N"	// DB 2105
VERSION : 0.0
  STRUCT
   Command_1_STATUS : WORD ;	//第1条命令的状态，0=正常，1=无响应，2=站号错误，3=命令错误，4=CRC校验错误
   Command_1_DATA_1 : WORD ;	//地址40021
   Command_1_DATA_2 : WORD ;	//地址40022
  END_STRUCT ;	
BEGIN
END_DATA_BLOCK

DATA_BLOCK DB 2111
VERSION : 0.0
  STRUCT
   START_SEQ : BYTE  := B#16#1;
   END_SEQ : BYTE  := B#16#2;
   SND_COMM_DB : WORD  := W#16#840;
   WRT_COMM_DB : WORD  := W#16#841;
   WRT_COMP_DB : WORD  := W#16#842;
   DAT_RECV_DB : WORD  := W#16#843;
   ACT_1 : BOOL  := TRUE;
   Mode_1 : BOOL ;
   SND_DB_1 : INT  := 2112;
   SND_ADD_1 : INT ;
   SND_LEN_1 : INT  := 6;
   RCV_DB_1 : INT  := 2115;
   RCV_ADD_1 : INT ;
   RCV_LEN_1 : INT  := 10;
   WD_TIME_1 : INT  := 3000;
   ACT_2 : BOOL  := TRUE;
   Mode_2 : BOOL ;
   SND_DB_2 : INT  := 2114;
   SND_ADD_2 : INT ;
   SND_LEN_2 : INT  := 10;
   RCV_DB_2 : INT  := 2115;
   RCV_ADD_2 : INT  := 10;
   RCV_LEN_2 : INT  := 2;
   WD_TIME_2 : INT  := 3000;
   VBVer : WORD  := W#16#29;	//配置文件版本号
  END_STRUCT ;	
BEGIN
   START_SEQ := B#16#1;
   END_SEQ := B#16#2;
   SND_COMM_DB := W#16#840;
   WRT_COMM_DB := W#16#841;
   WRT_COMP_DB := W#16#842;
   DAT_RECV_DB := W#16#843;
   ACT_1 := TRUE;
   SND_DB_1 := 2112;
   SND_LEN_1 := 6;
   RCV_DB_1 := 2115;
   RCV_LEN_1 := 10;
   WD_TIME_1 := 3000;
   ACT_2 := TRUE;
   SND_DB_2 := 2114;
   SND_LEN_2 := 10;
   RCV_DB_2 := 2115;
   RCV_ADD_2 := 10;
   RCV_LEN_2 := 2;
   WD_TIME_2 := 3000;
   VBVer := W#16#29;
END_DATA_BLOCK

DATA_BLOCK DB 2112
VERSION : 0.0
  STRUCT
   SlaveID_1 : BYTE  := B#16#B;
   FC_1 : BYTE  := B#16#3;
   START_ADD_1 : WORD ;
   DATA_NUM_1 : WORD  := W#16#4;
   CRC_1 : WORD ;
  END_STRUCT ;	
BEGIN
   SlaveID_1 := B#16#B;
   FC_1 := B#16#3;
   DATA_NUM_1 := W#16#4;
END_DATA_BLOCK

DATA_BLOCK "AP_FSB_WRITE"	// DB 2113
VERSION : 0.0
  STRUCT
   SlaveID_2 : BYTE  := B#16#B;
   FC_2 : BYTE  := B#16#10;
   START_ADD_2 : WORD  := W#16#4;
   DATA_NUM_2 : WORD  := W#16#1;
   DATA_BYTE_2 : WORD  := W#16#2;
   DATA_2_1 : WORD ;	//地址40005
   CRC_2 : WORD ;
  END_STRUCT ;	
BEGIN
   SlaveID_2 := B#16#B;
   FC_2 := B#16#10;
   START_ADD_2 := W#16#4;
   DATA_NUM_2 := W#16#1;
   DATA_BYTE_2 := W#16#2;
END_DATA_BLOCK

DATA_BLOCK DB 2114
VERSION : 0.0
  STRUCT
   SlaveID_2 : BYTE  := B#16#B;
   FC_2 : BYTE  := B#16#10;
   START_ADD_2 : WORD  := W#16#4;
   DATA_NUM_2 : WORD  := W#16#1;
   DATA_BYTE_2 : WORD  := W#16#2;
   DATA_NUM_2_1 : WORD ;
   CRC_2 : WORD ;
  END_STRUCT ;	
BEGIN
   SlaveID_2 := B#16#B;
   FC_2 := B#16#10;
   START_ADD_2 := W#16#4;
   DATA_NUM_2 := W#16#1;
   DATA_BYTE_2 := W#16#2;
END_DATA_BLOCK

DATA_BLOCK "AP_FSB_READ"	// DB 2115
VERSION : 0.0
  STRUCT
   Command_1_STATUS : WORD ;	//第1条命令的状态，0=正常，1=无响应，2=站号错误，3=命令错误，4=CRC校验错误
   Command_1_DATA_1 : WORD ;	//地址40001
   Command_1_DATA_2 : WORD ;	//地址40002
   Command_1_DATA_3 : WORD ;	//地址40003
   Command_1_DATA_4 : WORD ;	//地址40004
   Command_2_STATUS : WORD ;	//第2条命令的状态，0=正常，1=无响应，2=站号错误，3=命令错误，4=CRC校验错误
  END_STRUCT ;	
BEGIN
END_DATA_BLOCK

DATA_BLOCK DB 2121
VERSION : 0.0
  STRUCT
   START_SEQ : BYTE  := B#16#1;
   END_SEQ : BYTE  := B#16#2;
   SND_COMM_DB : WORD  := W#16#84A;
   WRT_COMM_DB : WORD  := W#16#84B;
   WRT_COMP_DB : WORD  := W#16#84C;
   DAT_RECV_DB : WORD  := W#16#84D;
   ACT_1 : BOOL  := TRUE;
   Mode_1 : BOOL ;
   SND_DB_1 : INT  := 2122;
   SND_ADD_1 : INT ;
   SND_LEN_1 : INT  := 6;
   RCV_DB_1 : INT  := 2125;
   RCV_ADD_1 : INT ;
   RCV_LEN_1 : INT  := 10;
   WD_TIME_1 : INT  := 3000;
   ACT_2 : BOOL  := TRUE;
   Mode_2 : BOOL ;
   SND_DB_2 : INT  := 2124;
   SND_ADD_2 : INT ;
   SND_LEN_2 : INT  := 10;
   RCV_DB_2 : INT  := 2125;
   RCV_ADD_2 : INT  := 10;
   RCV_LEN_2 : INT  := 2;
   WD_TIME_2 : INT  := 3000;
   VBVer : WORD  := W#16#29;	//配置文件版本号
  END_STRUCT ;	
BEGIN
   START_SEQ := B#16#1;
   END_SEQ := B#16#2;
   SND_COMM_DB := W#16#84A;
   WRT_COMM_DB := W#16#84B;
   WRT_COMP_DB := W#16#84C;
   DAT_RECV_DB := W#16#84D;
   ACT_1 := TRUE;
   SND_DB_1 := 2122;
   SND_LEN_1 := 6;
   RCV_DB_1 := 2125;
   RCV_LEN_1 := 10;
   WD_TIME_1 := 3000;
   ACT_2 := TRUE;
   SND_DB_2 := 2124;
   SND_LEN_2 := 10;
   RCV_DB_2 := 2125;
   RCV_ADD_2 := 10;
   RCV_LEN_2 := 2;
   WD_TIME_2 := 3000;
   VBVer := W#16#29;
END_DATA_BLOCK

DATA_BLOCK DB 2122
VERSION : 0.0
  STRUCT
   SlaveID_1 : BYTE  := B#16#B;
   FC_1 : BYTE  := B#16#3;
   START_ADD_1 : WORD ;
   DATA_NUM_1 : WORD  := W#16#4;
   CRC_1 : WORD ;
  END_STRUCT ;	
BEGIN
   SlaveID_1 := B#16#B;
   FC_1 := B#16#3;
   DATA_NUM_1 := W#16#4;
END_DATA_BLOCK

DATA_BLOCK "AT_QJSB_WRITE"	// DB 2123
VERSION : 0.0
  STRUCT
   SlaveID_2 : BYTE  := B#16#B;
   FC_2 : BYTE  := B#16#10;
   START_ADD_2 : WORD  := W#16#4;
   DATA_NUM_2 : WORD  := W#16#1;
   DATA_BYTE_2 : WORD  := W#16#2;
   DATA_2_1 : WORD ;	//地址40005
   CRC_2 : WORD ;
  END_STRUCT ;	
BEGIN
   SlaveID_2 := B#16#B;
   FC_2 := B#16#10;
   START_ADD_2 := W#16#4;
   DATA_NUM_2 := W#16#1;
   DATA_BYTE_2 := W#16#2;
END_DATA_BLOCK

DATA_BLOCK DB 2124
VERSION : 0.0
  STRUCT
   SlaveID_2 : BYTE  := B#16#B;
   FC_2 : BYTE  := B#16#10;
   START_ADD_2 : WORD  := W#16#4;
   DATA_NUM_2 : WORD  := W#16#1;
   DATA_BYTE_2 : WORD  := W#16#2;
   DATA_NUM_2_1 : WORD ;
   CRC_2 : WORD ;
  END_STRUCT ;	
BEGIN
   SlaveID_2 := B#16#B;
   FC_2 := B#16#10;
   START_ADD_2 := W#16#4;
   DATA_NUM_2 := W#16#1;
   DATA_BYTE_2 := W#16#2;
END_DATA_BLOCK

DATA_BLOCK "AT_QJSB_READ"	// DB 2125
VERSION : 0.0
  STRUCT
   Command_1_STATUS : WORD ;	//第1条命令的状态，0=正常，1=无响应，2=站号错误，3=命令错误，4=CRC校验错误
   Command_1_DATA_1 : WORD ;	//地址40001
   Command_1_DATA_2 : WORD ;	//地址40002
   Command_1_DATA_3 : WORD ;	//地址40003
   Command_1_DATA_4 : WORD ;	//地址40004
   Command_2_STATUS : WORD ;	//第2条命令的状态，0=正常，1=无响应，2=站号错误，3=命令错误，4=CRC校验错误
  END_STRUCT ;	
BEGIN
END_DATA_BLOCK

DATA_BLOCK "HF3_IMCC_Read_DB2291"	// DB 2291
VERSION : 0.1
  STRUCT
   IMCC_TO_BAS : WORD ;	//40001
   Fire_To_BAS : WORD ;	//40002
   Reserve_1 : ARRAY  [0 .. 3 ] OF WORD ;	//40003
   T6_XSF_A1_inRD : ARRAY  [0 .. 3 ] OF WORD  := W#16#0;	//40007
   Reserve_2 : ARRAY  [0 .. 3 ] OF WORD ;	//40011
   Reserve_3 : ARRAY  [0 .. 3 ] OF WORD ;	//40015
   K4_HPF_A1_inRD : ARRAY  [0 .. 3 ] OF WORD ;	//40019
   Reserve_4 : ARRAY  [0 .. 3 ] OF WORD  := W#16#0;	//40023
   T6_XPF_A1_inRD : ARRAY  [0 .. 3 ] OF WORD  := W#16#0;	//40027
   T7_XPF_A1 : ARRAY  [0 .. 3 ] OF WORD ;	//40031
   K4_XK_A1_inRD : ARRAY  [0 .. 3 ] OF WORD  := W#16#0;	//40035
   Reserve_5 : ARRAY  [0 .. 3 ] OF WORD ;	//40039
   Reserve_6 : ARRAY  [0 .. 3 ] OF WORD  := W#16#0;	//40043
   Reserve_7 : ARRAY  [0 .. 3 ] OF WORD ;	//40047
   Reserve_61 : ARRAY  [0 .. 3 ] OF WORD  := W#16#0;	//40051
   Reserve_62 : ARRAY  [0 .. 3 ] OF WORD  := W#16#0;
   Reserve_8 : ARRAY  [0 .. 3 ] OF WORD ;
   Reserve_9 : ARRAY  [0 .. 3 ] OF WORD ;	//40063
   Reserve_10 : ARRAY  [0 .. 3 ] OF WORD ;
   Reserve_11 : ARRAY  [0 .. 3 ] OF WORD ;	//40071
   Reserve_12 : ARRAY  [0 .. 103 ] OF WORD ;	//4075_40178
   TVF_A1_inRD : ARRAY  [0 .. 13 ] OF WORD  := W#16#0;	//40179
   TVF_A2_inRD : ARRAY  [0 .. 13 ] OF WORD  := W#16#0;	//40193
   Reserve_13 : ARRAY  [0 .. 13 ] OF WORD ;	//40207
   Reserve_14 : ARRAY  [0 .. 13 ] OF WORD ;
   UOF_A1_inRD : ARRAY  [0 .. 14 ] OF WORD  := W#16#0;	//40235
   Reserve_15 : ARRAY  [0 .. 14 ] OF WORD ;
   HPF_A1_inRD : ARRAY  [0 .. 7 ] OF WORD  := W#16#0;
   Reserve_16 : ARRAY  [0 .. 7 ] OF WORD  := W#16#0;
   KT_A1_inRD : ARRAY  [0 .. 10 ] OF WORD  := W#16#0;
   Reserve_17 : ARRAY  [0 .. 10 ] OF WORD  := W#16#0;	//40292
   K4_DTS_A1_inRD : WORD ;	//40303
   K4_DTS_A2_inRD : WORD ;
   K4_DTS_A3_inRD : WORD ;
   T6_D_A1_inRD : WORD ;
   T6_D_A2_inRD : WORD ;	//40307
   T7_D_A1_inRD : WORD ;
   T8_D_A1_inRD : WORD ;
   T8_D_A2_inRD : WORD ;
   Reserve_18 : ARRAY  [0 .. 15 ] OF WORD  := W#16#0;	//40311
   DM_A1_inRD : WORD ;	//40327
   DM_A2_inRD : WORD ;
   DM_A3_inRD : WORD ;
   DM_A4_inRD : WORD ;
   DM_A5_inRD : WORD ;
   DM_A6_inRD : WORD ;
   DM_A7_inRD : WORD ;
   DM_A8_inRD : WORD ;
   UOF_DTS_A1_inRD : WORD ;
   UOF_DTS_A2_inRD : WORD ;
   UOF_DTS_A3_inRD : WORD ;
   UOF_DTS_A4_inRD : WORD ;
   DTS_A1_inRD : WORD ;
   DTS_A2_inRD : WORD ;
   DTS_A3_inRD : WORD ;
   DTS_A4_inRD : WORD ;
   DTS_A5_inRD : WORD ;
   DTS_A6_inRD : WORD ;
   Reserve_21 : ARRAY  [0 .. 55 ] OF WORD  := W#16#0;	//40345
   LY1_inRD : WORD ;
   LY2_inRD : WORD ;
  END_STRUCT ;	
BEGIN
END_DATA_BLOCK

DATA_BLOCK "HF3_IMCC_Write_DB2292"	// DB 2292
VERSION : 0.1
  STRUCT
   BAS_To_IMCC : WORD ;	//40401
   Fire_To_IMCC : WORD ;
   Reserve_1 : WORD ;	//40403
   T6_XSF_A1_qnWR : WORD ;	//40404
   Reserve_2 : WORD ;
   Reserve_3 : WORD ;	//40406
   K4_HPF_A1_qnWR : WORD ;
   RFS_A_qnWR : WORD ;	//40408
   T6_XPF_A1_qnWR : WORD ;
   T7_XPF_A1_qnWR : WORD ;
   K4_XK_A1_qnWR : WORD ;	//40411
   Reserve_4 : WORD ;
   Reserve_5 : WORD ;	//40413
   Reserve_6 : WORD ;
   Reserve_61 : WORD ;
   Reserve_62 : WORD ;	//40416
   Reserve_8 : ARRAY  [0 .. 29 ] OF WORD ;
   TVF_A1_qnWR : WORD ;	//40447
   TVF_A2_qnWR : WORD ;
   Reserve_9 : ARRAY  [0 .. 1 ] OF WORD ;
   UOF_A1_qnWR : ARRAY  [0 .. 1 ] OF WORD ;	//40451
   Reserve_10 : ARRAY  [0 .. 1 ] OF WORD ;
   HPF_A1_qnWR : ARRAY  [0 .. 1 ] OF WORD ;	//40455
   Reserve_11 : ARRAY  [0 .. 1 ] OF WORD ;
   KT_A1_qnWR : ARRAY  [0 .. 1 ] OF WORD ;	//40459
   Reserve_12 : ARRAY  [0 .. 1 ] OF WORD ;
   K4_DTS_A1_qnWR : WORD ;	//40463
   K4_DTS_A2_qnWR : WORD ;
   K4_DTS_A3_qnWR : WORD ;
   T6_D_A1_qnWR : WORD ;
   T6_D_A2_qnWR : WORD ;
   T7_D_A1_qnWR : WORD ;
   T8_D_A1_qnWR : WORD ;
   T8_D_A2_qnWR : WORD ;
   Reserve_14 : ARRAY  [0 .. 15 ] OF WORD ;	//40471
   DM_A1_qnWR : WORD ;
   DM_A2_qnWR : WORD ;
   DM_A3_qnWR : WORD ;
   DM_A4_qnWR : WORD ;
   DM_A5_qnWR : WORD ;
   DM_A6_qnWR : WORD ;
   DM_A7_qnWR : WORD ;
   DM_A8_qnWR : WORD ;
   UOF_DTS_A1_qnWR : WORD ;
   UOF_DTS_A2_qnWR : WORD ;
   UOF_DTS_A3_qnWR : WORD ;
   UOF_DTS_A4_qnWR : WORD ;
   DTS_A1_qnWR : WORD ;	//40499
   DTS_A2_qnWR : WORD ;
   DTS_A3_qnWR : WORD ;
   DTS_A4_qnWR : WORD ;
   DTS_A5_qnWR : WORD ;
   DTS_A6_qnWR : WORD ;
   Reserve_15 : ARRAY  [0 .. 55 ] OF WORD ;
   LY1_inRD : WORD ;
   LY2_inRD : WORD ;
  END_STRUCT ;	
BEGIN
END_DATA_BLOCK

DATA_BLOCK DB 2351
VERSION : 0.0
  STRUCT
   START_SEQ : BYTE  := B#16#1;
   END_SEQ : BYTE  := B#16#1;
   SND_COMM_DB : WORD  := W#16#930;
   WRT_COMM_DB : WORD  := W#16#931;
   WRT_COMP_DB : WORD  := W#16#932;
   DAT_RECV_DB : WORD  := W#16#933;
   ACT_1 : BOOL  := TRUE;
   Mode_1 : BOOL ;
   SND_DB_1 : INT  := 2352;
   SND_ADD_1 : INT ;
   SND_LEN_1 : INT  := 6;
   RCV_DB_1 : INT  := 2355;
   RCV_ADD_1 : INT ;
   RCV_LEN_1 : INT  := 4;
   WD_TIME_1 : INT  := 3000;
  END_STRUCT ;	
BEGIN
   START_SEQ := B#16#1;
   END_SEQ := B#16#1;
   SND_COMM_DB := W#16#930;
   WRT_COMM_DB := W#16#931;
   WRT_COMP_DB := W#16#932;
   DAT_RECV_DB := W#16#933;
   ACT_1 := TRUE;
   SND_DB_1 := 2352;
   SND_LEN_1 := 6;
   RCV_DB_1 := 2355;
   RCV_LEN_1 := 4;
   WD_TIME_1 := 3000;
END_DATA_BLOCK

DATA_BLOCK DB 2352
VERSION : 0.0
  STRUCT
   SlaveID_1 : BYTE  := B#16#B;
   FC_1 : BYTE  := B#16#3;
   START_ADD_1 : WORD ;
   DATA_NUM_1 : WORD  := W#16#1;
   CRC_1 : WORD ;
  END_STRUCT ;	
BEGIN
   SlaveID_1 := B#16#B;
   FC_1 := B#16#3;
   DATA_NUM_1 := W#16#1;
END_DATA_BLOCK

DATA_BLOCK DB 2355
VERSION : 0.0
  STRUCT
   Command_1_STATUS : WORD ;	//第1条命令的状态，0=正常，1=无响应，2=站号错误，3=命令错误，4=CRC校验错误
   Command_1_DATA_1 : WORD ;	//地址40001
  END_STRUCT ;	
BEGIN
END_DATA_BLOCK

DATA_BLOCK "HF3_EPS_HMI"	// DB 2501
VERSION : 0.0
"HF3_EPS_FB2501"
BEGIN
END_DATA_BLOCK

DATA_BLOCK DB 2552
VERSION : 0.0
"HF3_IMCC_CommOK_FB2512"
BEGIN
END_DATA_BLOCK

DATA_BLOCK "IMCC_LOCK"	// DB 2555
VERSION : 0.1
  STRUCT
   KT_A1_Stop : BOOL ;
   HPF_A1_Stop : BOOL ;
   DTS_A1_Open : BOOL ;
   DTS_A2_Open : BOOL ;
   DTS_A3_Open : BOOL ;
   DTS_A4_Open : BOOL ;
   DTS_A5_Open : BOOL ;
   DTS_A6_Open : BOOL ;
   TVF_A1_Stop : BOOL ;
   TVF_A2_Stop : BOOL ;
   UOF_A1_Stop : BOOL ;
   DM_A1_Open : BOOL ;
   DM_A2_Open : BOOL ;
   DM_A3_Open : BOOL ;
   DM_A4_Open : BOOL ;
   DM_A5_Open : BOOL ;
   DM_A6_Open : BOOL ;
   DM_A7_Open : BOOL ;
   DM_A8_Open : BOOL ;
   U0F_DT_A1_Open : BOOL ;
   U0F_DT_A2_Open : BOOL ;
   U0F_DT_A3_Open : BOOL ;
   U0F_DT_A4_Open : BOOL ;
   K4_XK_A1_Stop : BOOL ;
   K4_HPF_A1_Stop : BOOL ;
   K4_DT_A1_Open : BOOL ;
   K4_DT_A2_Open : BOOL ;
   K4_DT_A3_Open : BOOL ;
   T6_XPF_A1_Stop : BOOL ;
   T6_XSF_A1_Stop : BOOL ;
   T6_D_A1_Open : BOOL ;
   T6_D_A2_Open : BOOL ;
   T7_XPF_A1_Stop : BOOL ;
   T7_D_A1_Open : BOOL ;
  END_STRUCT ;	
BEGIN
END_DATA_BLOCK

DATA_BLOCK DB 2592
VERSION : 0.0
"HF3_PSB_FB2591"
BEGIN
END_DATA_BLOCK

DATA_BLOCK DB 2602
VERSION : 0.0
"HF3_LSQK_FB2521"
BEGIN
END_DATA_BLOCK

DATA_BLOCK DB 2652
VERSION : 0.0
"HF3_JET_FB2531"
BEGIN
END_DATA_BLOCK

DATA_BLOCK DB 2702
VERSION : 0.0
"HF3_VRV_FB2541"
BEGIN
END_DATA_BLOCK

DATA_BLOCK DB 2752
VERSION : 0.0
"HF3_SB_FB2551"
BEGIN
END_DATA_BLOCK

DATA_BLOCK DB 2802
VERSION : 0.0
"HF3_3#SB_FB2561"
BEGIN
END_DATA_BLOCK

DATA_BLOCK DB 2821
VERSION : 0.0
"HF3_Senor_FB2821"
BEGIN
END_DATA_BLOCK

DATA_BLOCK DB 2952
VERSION : 0.0
FB 2571
BEGIN
END_DATA_BLOCK

DATA_BLOCK DB 3007
VERSION : 0.0
FB 3007
BEGIN
END_DATA_BLOCK

DATA_BLOCK DB 3052
VERSION : 0.0
"HF3_UPS_FB2611"
BEGIN
END_DATA_BLOCK

DATA_BLOCK DB 3102
VERSION : 0.0
"HF3_DT_FB2621"
BEGIN
END_DATA_BLOCK

DATA_BLOCK DB 3152
VERSION : 0.0
"HF3_FT_FB2631"
BEGIN
END_DATA_BLOCK

DATA_BLOCK DB 3252
VERSION : 0.0
"HF3_IMCC_TVF_FB2651"
BEGIN
END_DATA_BLOCK

DATA_BLOCK DB 3302
VERSION : 0.0
"HF3_IMCC_TEF_FB2661"
BEGIN
END_DATA_BLOCK

DATA_BLOCK DB 3352
VERSION : 0.0
"HF3_IMCC_KT_FB2671"
BEGIN
END_DATA_BLOCK

DATA_BLOCK DB 3402
VERSION : 0.0
"HF3_IMCC_HPF_FB2681"
BEGIN
END_DATA_BLOCK

DATA_BLOCK DB 3452
VERSION : 0.0
"HF3_IMCC_FJ_FB2691"
BEGIN
END_DATA_BLOCK

DATA_BLOCK DB 3502
VERSION : 0.0
"HF3_IMCC_DZ_FB2701"
BEGIN
END_DATA_BLOCK

DATA_BLOCK DB 3552
VERSION : 0.0
"HF3_IMCC_DT_FB2711"
BEGIN
END_DATA_BLOCK

DATA_BLOCK DB 3602
VERSION : 0.0
"HF3_IMCC_D_FB2721"
BEGIN
END_DATA_BLOCK

DATA_BLOCK DB 3652
VERSION : 0.0
"HF3_JH_YC_FB2731"
BEGIN
END_DATA_BLOCK

DATA_BLOCK DB 3752
VERSION : 0.0
"HF3_DPH_FB2751"
BEGIN
END_DATA_BLOCK

DATA_BLOCK DB 3802
VERSION : 0.0
"HF3_FJ_FB2761"
BEGIN
END_DATA_BLOCK

DATA_BLOCK DB 4002
VERSION : 0.0
"HF3_FJPG_FB2771"
BEGIN
END_DATA_BLOCK

DATA_BLOCK DB 4052
VERSION : 0.0
"HF3_XFDF_FB2781"
BEGIN
END_DATA_BLOCK

DATA_BLOCK DB 4102
VERSION : 0.0
"HF3_EPS_WLE_FB2791"
BEGIN
END_DATA_BLOCK

DATA_BLOCK DB 4151
VERSION : 0.0
"HF3_D_FB2801"
BEGIN
END_DATA_BLOCK

DATA_BLOCK DB 4202
VERSION : 0.0
"HF3_FHF_RFM_FB2811"
BEGIN
END_DATA_BLOCK

DATA_BLOCK DB 4251
VERSION : 0.0
"HF3_Senor_FB2821"
BEGIN
END_DATA_BLOCK

DATA_BLOCK DB 4302
VERSION : 0.0
"从端与主端通讯"
BEGIN
END_DATA_BLOCK

